// TIA Portal V17 export
// export: Created 2025-03-07T09:18:59.1372359Z, ExportSetting WithDefaults, DisplayName Totally Integrated Automation Portal, DisplayVersion V17 Update 8, DisplayName TIA Portal Openness, DisplayVersion V17 Update 8, DisplayName TIA Portal Version Control Interface, DisplayVersion V17, DisplayName SINAMICS Startdrive Advanced, DisplayVersion V17 SP2, DisplayName SINAMICS Startdrive G110M, G120, G120C, G120D, G120P, G115D, DisplayVersion V17 SP2, DisplayName SINAMICS Startdrive G130, G150, S120, S150, SINAMICS MV, S210, DisplayVersion V17 SP2, DisplayName STEP 7 Professional, DisplayVersion V17 Update 8, DisplayName SINUMERIK ONE STEP 7 Toolbox, DisplayVersion V17 Update 12, DisplayName SINUMERIK 840D sl STEP 7 Toolbox, DisplayVersion V17 Update 12, DisplayName STEP 7 Safety, DisplayVersion V17 Update 6, DisplayName WinCC Advanced, DisplayVersion V17 Update 8
FUNCTION "FC16017_METHOD_CALLS_U03_MEAS_STA_MEAS_B" : Void   // FC16017, LAD
{ S7_Optimized_Access := 'TRUE' }
VERSION : 0.1
// stored: AutoNumber false, IsIECCheckEnabled false, SetENOAutomatically false, UDAEnableTagReadback false
   VAR_TEMP
      AUX_WSTRING_PART_ID_MEAS_STA : WString;
      AUX_WCHARS : Array[0..63] of WChar;
      index : Int;
      AUX_ALARMS : Bool;
   END_VAR
   VAR_TEMP   // added for the SCL form of the ladder/FBD networks
      _w1 : Bool;
      _w2 : Bool;
   END_VAR
BEGIN

REGION Network 1 (SCL): TRANSFORM TO WCHARS
   FOR #index := 0 TO 63 DO
       #AUX_WCHARS[#index] := CHAR_TO_WCHAR("DB8000_PART_STATUS".UNIT_03.FIXTURE_1.PART_A.PART_ID[#index]);
   END_FOR;
END_REGION

REGION Network 2: TRANSFORM TO WSTRING
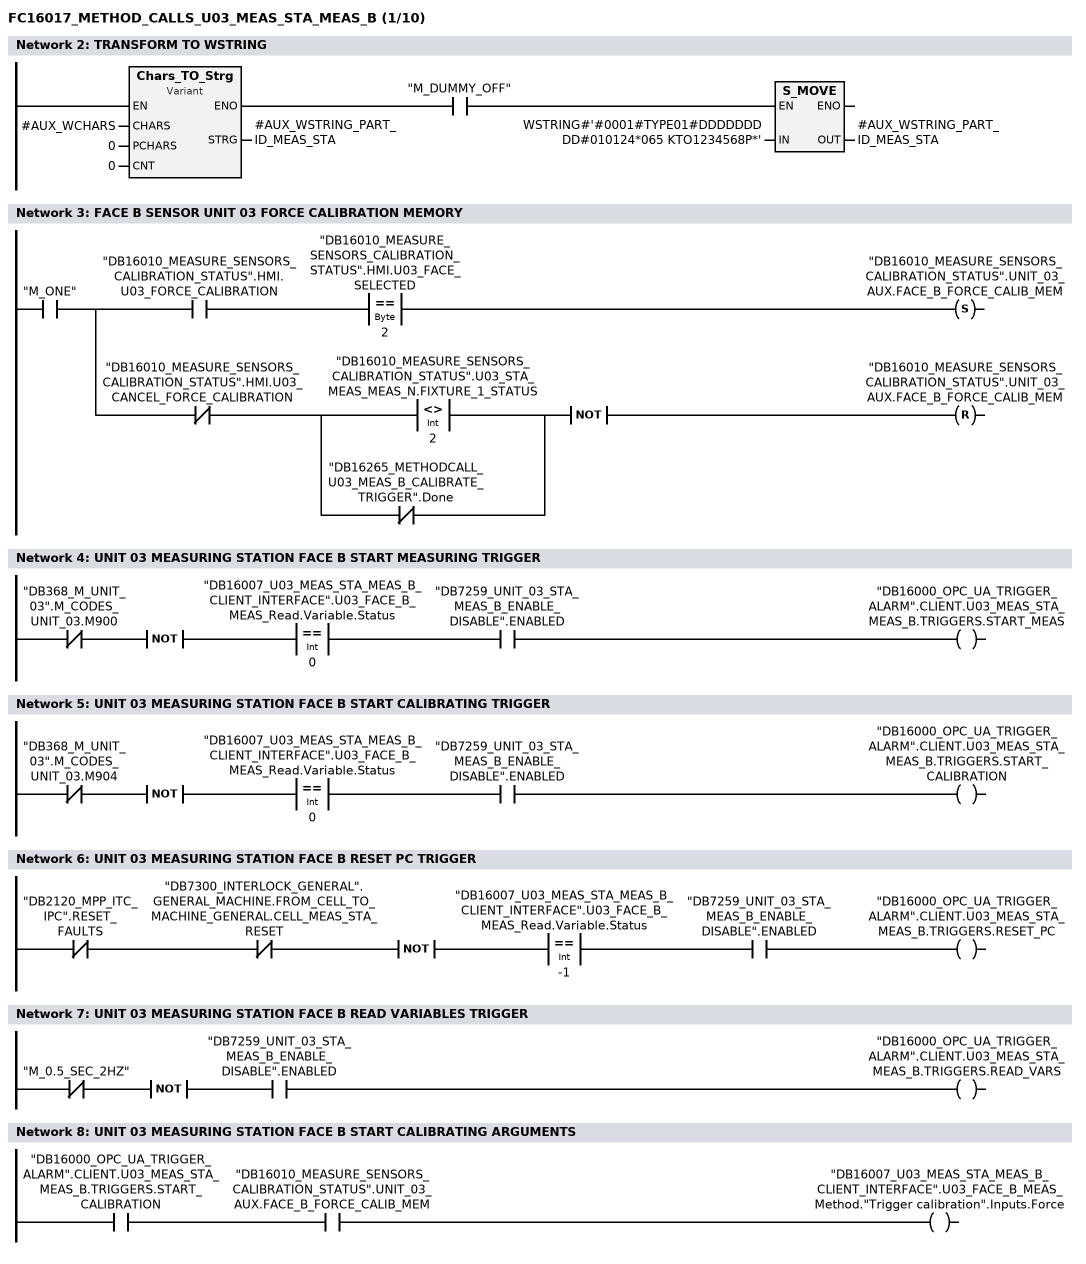
   RUNG wire#powerrail
      { S7_Templates := "[ptr_type := Variant, str_type := WString]" } Chars_TO_Strg(Chars := #AUX_WCHARS, pChars := 0, Cnt := 0, Strg => #AUX_WSTRING_PART_ID_MEAS_STA)
      Contact( "M_DUMMY_OFF" )
      S_Move(in := WSTRING#'#0001#TYPE01#DDDDDDDDD#010124*065 KTO1234568P*', out => #AUX_WSTRING_PART_ID_MEAS_STA)
   END_RUNG
   // the same network as SCL:
   Chars_TO_Strg(Chars := #AUX_WCHARS,
                 pChars := 0,
                 Cnt := 0,
                 Strg => #AUX_WSTRING_PART_ID_MEAS_STA,
                 ENO => #_w1);
   IF #_w1 AND "M_DUMMY_OFF" THEN
       #AUX_WSTRING_PART_ID_MEAS_STA := WSTRING#'#0001#TYPE01#DDDDDDDDD#010124*065 KTO1234568P*';
   END_IF;
END_REGION

REGION Network 3: FACE B SENSOR UNIT 03 FORCE CALIBRATION MEMORY
   RUNG wire#powerrail
      Contact( "M_ONE" )
      wire#w1
      Contact( "DB16010_MEASURE_SENSORS_CALIBRATION_STATUS".HMI.U03_FORCE_CALIBRATION )
      { S7_Templates := "SrcType := Byte" } EQ_Contact(in1 := "DB16010_MEASURE_SENSORS_CALIBRATION_STATUS".HMI.U03_FACE_SELECTED, in2 := 2)
      S_Coil( "DB16010_MEASURE_SENSORS_CALIBRATION_STATUS".UNIT_03_AUX.FACE_B_FORCE_CALIB_MEM )
   END_RUNG
   RUNG wire#w1
      I_Contact( "DB16010_MEASURE_SENSORS_CALIBRATION_STATUS".HMI.U03_CANCEL_FORCE_CALIBRATION )
      wire#w2
      { S7_Templates := "SrcType := Int" } NE_Contact(in1 := "DB16010_MEASURE_SENSORS_CALIBRATION_STATUS".U03_STA_MEAS_MEAS_N.FIXTURE_1_STATUS, in2 := 2)
      wire#w3
      Not()
      R_Coil( "DB16010_MEASURE_SENSORS_CALIBRATION_STATUS".UNIT_03_AUX.FACE_B_FORCE_CALIB_MEM )
   END_RUNG
   RUNG wire#w2
      I_Contact( "DB16265_METHODCALL_U03_MEAS_B_CALIBRATE_TRIGGER".Done )
   END_RUNG wire#w3
   // the same network as SCL:
   IF "M_ONE" AND "DB16010_MEASURE_SENSORS_CALIBRATION_STATUS".HMI.U03_FORCE_CALIBRATION AND ("DB16010_MEASURE_SENSORS_CALIBRATION_STATUS".HMI.U03_FACE_SELECTED = 2) THEN
       "DB16010_MEASURE_SENSORS_CALIBRATION_STATUS".UNIT_03_AUX.FACE_B_FORCE_CALIB_MEM := TRUE;
   END_IF;
   IF NOT ("M_ONE" AND NOT "DB16010_MEASURE_SENSORS_CALIBRATION_STATUS".HMI.U03_CANCEL_FORCE_CALIBRATION AND (("DB16010_MEASURE_SENSORS_CALIBRATION_STATUS".U03_STA_MEAS_MEAS_N.FIXTURE_1_STATUS <> 2) OR NOT "DB16265_METHODCALL_U03_MEAS_B_CALIBRATE_TRIGGER".Done)) THEN
       "DB16010_MEASURE_SENSORS_CALIBRATION_STATUS".UNIT_03_AUX.FACE_B_FORCE_CALIB_MEM := FALSE;
   END_IF;
END_REGION

REGION Network 4: UNIT 03 MEASURING STATION FACE B START MEASURING TRIGGER
   RUNG wire#powerrail
      I_Contact( "DB368_M_UNIT_03".M_CODES_UNIT_03.M900 )
      Not()
      { S7_Templates := "SrcType := Int" } EQ_Contact(in1 := "DB16007_U03_MEAS_STA_MEAS_B_CLIENT_INTERFACE".U03_FACE_B_MEAS_Read.Variable.Status, in2 := 0)
      Contact( "DB7259_UNIT_03_STA_MEAS_B_ENABLE_DISABLE".ENABLED )
      Coil( "DB16000_OPC_UA_TRIGGER_ALARM".CLIENT.U03_MEAS_STA_MEAS_B.TRIGGERS.START_MEAS )
   END_RUNG
   // the same network as SCL:
   "DB16000_OPC_UA_TRIGGER_ALARM".CLIENT.U03_MEAS_STA_MEAS_B.TRIGGERS.START_MEAS := NOT (NOT "DB368_M_UNIT_03".M_CODES_UNIT_03.M900) AND ("DB16007_U03_MEAS_STA_MEAS_B_CLIENT_INTERFACE".U03_FACE_B_MEAS_Read.Variable.Status = 0) AND "DB7259_UNIT_03_STA_MEAS_B_ENABLE_DISABLE".ENABLED;
END_REGION

REGION Network 5: UNIT 03 MEASURING STATION FACE B START CALIBRATING TRIGGER
   RUNG wire#powerrail
      I_Contact( "DB368_M_UNIT_03".M_CODES_UNIT_03.M904 )
      Not()
      { S7_Templates := "SrcType := Int" } EQ_Contact(in1 := "DB16007_U03_MEAS_STA_MEAS_B_CLIENT_INTERFACE".U03_FACE_B_MEAS_Read.Variable.Status, in2 := 0)
      Contact( "DB7259_UNIT_03_STA_MEAS_B_ENABLE_DISABLE".ENABLED )
      Coil( "DB16000_OPC_UA_TRIGGER_ALARM".CLIENT.U03_MEAS_STA_MEAS_B.TRIGGERS.START_CALIBRATION )
   END_RUNG
   // the same network as SCL:
   "DB16000_OPC_UA_TRIGGER_ALARM".CLIENT.U03_MEAS_STA_MEAS_B.TRIGGERS.START_CALIBRATION := NOT (NOT "DB368_M_UNIT_03".M_CODES_UNIT_03.M904) AND ("DB16007_U03_MEAS_STA_MEAS_B_CLIENT_INTERFACE".U03_FACE_B_MEAS_Read.Variable.Status = 0) AND "DB7259_UNIT_03_STA_MEAS_B_ENABLE_DISABLE".ENABLED;
END_REGION

REGION Network 6: UNIT 03 MEASURING STATION FACE B RESET PC TRIGGER
   RUNG wire#powerrail
      I_Contact( "DB2120_MPP_ITC_IPC".RESET_FAULTS )
      I_Contact( "DB7300_INTERLOCK_GENERAL".GENERAL_MACHINE.FROM_CELL_TO_MACHINE_GENERAL.CELL_MEAS_STA_RESET )
      Not()
      { S7_Templates := "SrcType := Int" } EQ_Contact(in1 := "DB16007_U03_MEAS_STA_MEAS_B_CLIENT_INTERFACE".U03_FACE_B_MEAS_Read.Variable.Status, in2 := -1)
      Contact( "DB7259_UNIT_03_STA_MEAS_B_ENABLE_DISABLE".ENABLED )
      Coil( "DB16000_OPC_UA_TRIGGER_ALARM".CLIENT.U03_MEAS_STA_MEAS_B.TRIGGERS.RESET_PC )
   END_RUNG
   // the same network as SCL:
   "DB16000_OPC_UA_TRIGGER_ALARM".CLIENT.U03_MEAS_STA_MEAS_B.TRIGGERS.RESET_PC := NOT (NOT "DB2120_MPP_ITC_IPC".RESET_FAULTS AND NOT "DB7300_INTERLOCK_GENERAL".GENERAL_MACHINE.FROM_CELL_TO_MACHINE_GENERAL.CELL_MEAS_STA_RESET) AND ("DB16007_U03_MEAS_STA_MEAS_B_CLIENT_INTERFACE".U03_FACE_B_MEAS_Read.Variable.Status = (-1)) AND "DB7259_UNIT_03_STA_MEAS_B_ENABLE_DISABLE".ENABLED;
END_REGION

REGION Network 7: UNIT 03 MEASURING STATION FACE B READ VARIABLES TRIGGER
   RUNG wire#powerrail
      I_Contact( "M_0.5_SEC_2HZ" )
      Not()
      Contact( "DB7259_UNIT_03_STA_MEAS_B_ENABLE_DISABLE".ENABLED )
      Coil( "DB16000_OPC_UA_TRIGGER_ALARM".CLIENT.U03_MEAS_STA_MEAS_B.TRIGGERS.READ_VARS )
   END_RUNG
   // the same network as SCL:
   "DB16000_OPC_UA_TRIGGER_ALARM".CLIENT.U03_MEAS_STA_MEAS_B.TRIGGERS.READ_VARS := NOT (NOT "M_0.5_SEC_2HZ") AND "DB7259_UNIT_03_STA_MEAS_B_ENABLE_DISABLE".ENABLED;
END_REGION

REGION Network 8: UNIT 03 MEASURING STATION FACE B START CALIBRATING ARGUMENTS
   RUNG wire#powerrail
      Contact( "DB16000_OPC_UA_TRIGGER_ALARM".CLIENT.U03_MEAS_STA_MEAS_B.TRIGGERS.START_CALIBRATION )
      Contact( "DB16010_MEASURE_SENSORS_CALIBRATION_STATUS".UNIT_03_AUX.FACE_B_FORCE_CALIB_MEM )
      Coil( "DB16007_U03_MEAS_STA_MEAS_B_CLIENT_INTERFACE".U03_FACE_B_MEAS_Method."Trigger calibration".Inputs.Force )
   END_RUNG
   // the same network as SCL:
   "DB16007_U03_MEAS_STA_MEAS_B_CLIENT_INTERFACE".U03_FACE_B_MEAS_Method."Trigger calibration".Inputs.Force := "DB16000_OPC_UA_TRIGGER_ALARM".CLIENT.U03_MEAS_STA_MEAS_B.TRIGGERS.START_CALIBRATION AND "DB16010_MEASURE_SENSORS_CALIBRATION_STATUS".UNIT_03_AUX.FACE_B_FORCE_CALIB_MEM;
END_REGION

REGION Network 9: UNIT 03 MEASURING STATION FACE B START MEASURING TRIGGER CALL
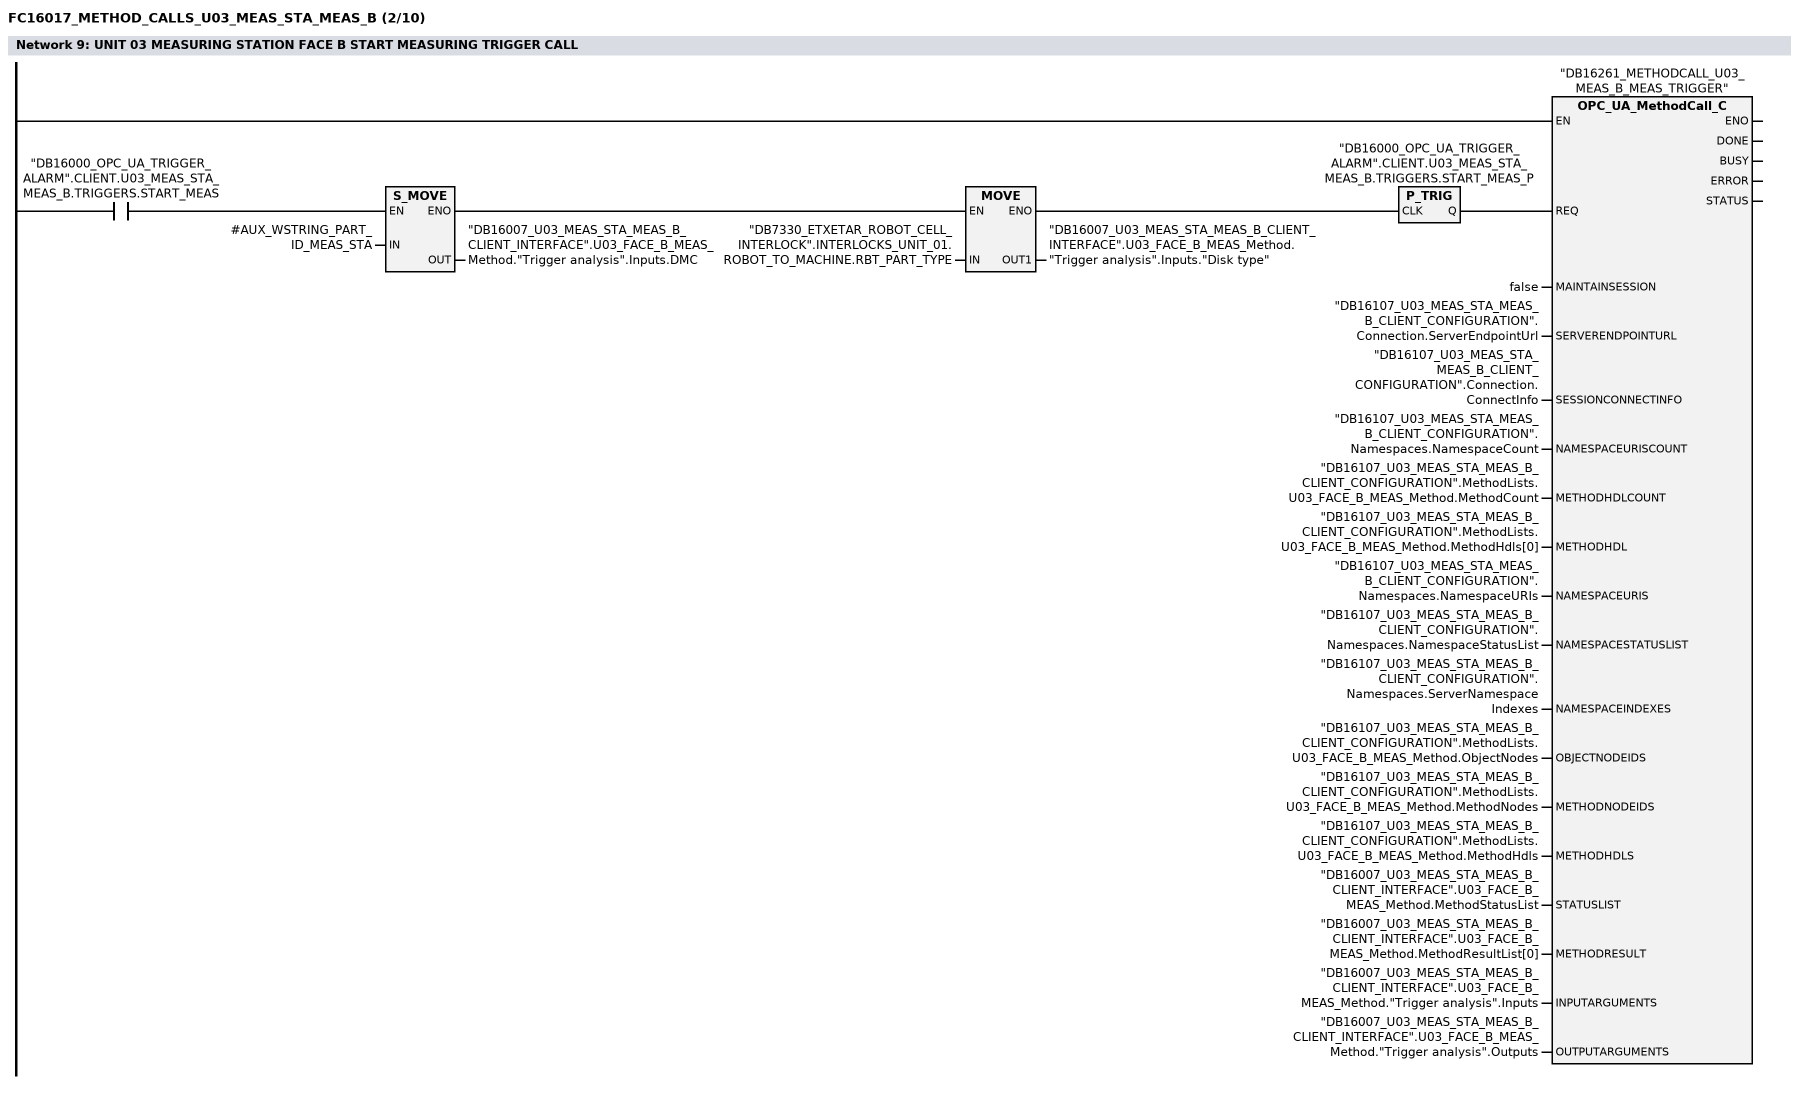
   RUNG wire#powerrail
      "DB16261_METHODCALL_U03_MEAS_B_MEAS_TRIGGER".OPC_UA_MethodCall_C(REQ := wire#w1, MaintainSession := false, ServerEndpointUrl := "DB16107_U03_MEAS_STA_MEAS_B_CLIENT_CONFIGURATION".Connection.ServerEndpointUrl, SessionConnectInfo := "DB16107_U03_MEAS_STA_MEAS_B_CLIENT_CONFIGURATION".Connection.ConnectInfo, NamespaceUrisCount := "DB16107_U03_MEAS_STA_MEAS_B_CLIENT_CONFIGURATION".Namespaces.NamespaceCount, MethodHdlCount := "DB16107_U03_MEAS_STA_MEAS_B_CLIENT_CONFIGURATION".MethodLists.U03_FACE_B_MEAS_Method.MethodCount, MethodHdl := "DB16107_U03_MEAS_STA_MEAS_B_CLIENT_CONFIGURATION".MethodLists.U03_FACE_B_MEAS_Method.MethodHdls[0], NamespaceUris := "DB16107_U03_MEAS_STA_MEAS_B_CLIENT_CONFIGURATION".Namespaces.NamespaceURIs, NamespaceStatusList := "DB16107_U03_MEAS_STA_MEAS_B_CLIENT_CONFIGURATION".Namespaces.NamespaceStatusList, NamespaceIndexes := "DB16107_U03_MEAS_STA_MEAS_B_CLIENT_CONFIGURATION".Namespaces.ServerNamespaceIndexes, ObjectNodeIDs := "DB16107_U03_MEAS_STA_MEAS_B_CLIENT_CONFIGURATION".MethodLists.U03_FACE_B_MEAS_Method.ObjectNodes, MethodNodeIDs := "DB16107_U03_MEAS_STA_MEAS_B_CLIENT_CONFIGURATION".MethodLists.U03_FACE_B_MEAS_Method.MethodNodes, MethodHdls := "DB16107_U03_MEAS_STA_MEAS_B_CLIENT_CONFIGURATION".MethodLists.U03_FACE_B_MEAS_Method.MethodHdls, StatusList := "DB16007_U03_MEAS_STA_MEAS_B_CLIENT_INTERFACE".U03_FACE_B_MEAS_Method.MethodStatusList, MethodResult := "DB16007_U03_MEAS_STA_MEAS_B_CLIENT_INTERFACE".U03_FACE_B_MEAS_Method.MethodResultList[0], InputArguments := "DB16007_U03_MEAS_STA_MEAS_B_CLIENT_INTERFACE".U03_FACE_B_MEAS_Method."Trigger analysis".Inputs, OutputArguments := "DB16007_U03_MEAS_STA_MEAS_B_CLIENT_INTERFACE".U03_FACE_B_MEAS_Method."Trigger analysis".Outputs, Done =>, Busy =>, Error =>, Status =>)
   END_RUNG
   RUNG wire#powerrail
      Contact( "DB16000_OPC_UA_TRIGGER_ALARM".CLIENT.U03_MEAS_STA_MEAS_B.TRIGGERS.START_MEAS )
      S_Move(in := #AUX_WSTRING_PART_ID_MEAS_STA, out => "DB16007_U03_MEAS_STA_MEAS_B_CLIENT_INTERFACE".U03_FACE_B_MEAS_Method."Trigger analysis".Inputs.DMC)
      Move(in := "DB7330_ETXETAR_ROBOT_CELL_INTERLOCK".INTERLOCKS_UNIT_01.ROBOT_TO_MACHINE.RBT_PART_TYPE, out1 => "DB16007_U03_MEAS_STA_MEAS_B_CLIENT_INTERFACE".U03_FACE_B_MEAS_Method."Trigger analysis".Inputs."Disk type")
      P_Trig( "DB16000_OPC_UA_TRIGGER_ALARM".CLIENT.U03_MEAS_STA_MEAS_B.TRIGGERS.START_MEAS_P )
   END_RUNG wire#w1
   // the same network as SCL:
   IF "DB16000_OPC_UA_TRIGGER_ALARM".CLIENT.U03_MEAS_STA_MEAS_B.TRIGGERS.START_MEAS THEN
       "DB16007_U03_MEAS_STA_MEAS_B_CLIENT_INTERFACE".U03_FACE_B_MEAS_Method."Trigger analysis".Inputs.DMC := #AUX_WSTRING_PART_ID_MEAS_STA;
       "DB16007_U03_MEAS_STA_MEAS_B_CLIENT_INTERFACE".U03_FACE_B_MEAS_Method."Trigger analysis".Inputs."Disk type" := "DB7330_ETXETAR_ROBOT_CELL_INTERLOCK".INTERLOCKS_UNIT_01.ROBOT_TO_MACHINE.RBT_PART_TYPE;
   END_IF;
   #_w1 := "DB16000_OPC_UA_TRIGGER_ALARM".CLIENT.U03_MEAS_STA_MEAS_B.TRIGGERS.START_MEAS AND NOT "DB16000_OPC_UA_TRIGGER_ALARM".CLIENT.U03_MEAS_STA_MEAS_B.TRIGGERS.START_MEAS_P;   // rising edge
   "DB16000_OPC_UA_TRIGGER_ALARM".CLIENT.U03_MEAS_STA_MEAS_B.TRIGGERS.START_MEAS_P := "DB16000_OPC_UA_TRIGGER_ALARM".CLIENT.U03_MEAS_STA_MEAS_B.TRIGGERS.START_MEAS;
   "DB16261_METHODCALL_U03_MEAS_B_MEAS_TRIGGER"(REQ := #_w1,   // OPC_UA_MethodCall_C
                           MaintainSession := false,
                           ServerEndpointUrl := "DB16107_U03_MEAS_STA_MEAS_B_CLIENT_CONFIGURATION".Connection.ServerEndpointUrl,
                           SessionConnectInfo := "DB16107_U03_MEAS_STA_MEAS_B_CLIENT_CONFIGURATION".Connection.ConnectInfo,
                           NamespaceUrisCount := "DB16107_U03_MEAS_STA_MEAS_B_CLIENT_CONFIGURATION".Namespaces.NamespaceCount,
                           MethodHdlCount := "DB16107_U03_MEAS_STA_MEAS_B_CLIENT_CONFIGURATION".MethodLists.U03_FACE_B_MEAS_Method.MethodCount,
                           MethodHdl := "DB16107_U03_MEAS_STA_MEAS_B_CLIENT_CONFIGURATION".MethodLists.U03_FACE_B_MEAS_Method.MethodHdls[0],
                           NamespaceUris := "DB16107_U03_MEAS_STA_MEAS_B_CLIENT_CONFIGURATION".Namespaces.NamespaceURIs,
                           NamespaceStatusList := "DB16107_U03_MEAS_STA_MEAS_B_CLIENT_CONFIGURATION".Namespaces.NamespaceStatusList,
                           NamespaceIndexes := "DB16107_U03_MEAS_STA_MEAS_B_CLIENT_CONFIGURATION".Namespaces.ServerNamespaceIndexes,
                           ObjectNodeIDs := "DB16107_U03_MEAS_STA_MEAS_B_CLIENT_CONFIGURATION".MethodLists.U03_FACE_B_MEAS_Method.ObjectNodes,
                           MethodNodeIDs := "DB16107_U03_MEAS_STA_MEAS_B_CLIENT_CONFIGURATION".MethodLists.U03_FACE_B_MEAS_Method.MethodNodes,
                           MethodHdls := "DB16107_U03_MEAS_STA_MEAS_B_CLIENT_CONFIGURATION".MethodLists.U03_FACE_B_MEAS_Method.MethodHdls,
                           StatusList := "DB16007_U03_MEAS_STA_MEAS_B_CLIENT_INTERFACE".U03_FACE_B_MEAS_Method.MethodStatusList,
                           MethodResult := "DB16007_U03_MEAS_STA_MEAS_B_CLIENT_INTERFACE".U03_FACE_B_MEAS_Method.MethodResultList[0],
                           InputArguments := "DB16007_U03_MEAS_STA_MEAS_B_CLIENT_INTERFACE".U03_FACE_B_MEAS_Method."Trigger analysis".Inputs,
                           OutputArguments := "DB16007_U03_MEAS_STA_MEAS_B_CLIENT_INTERFACE".U03_FACE_B_MEAS_Method."Trigger analysis".Outputs);
END_REGION

REGION Network 10: UNIT 03 MEASURING STATION FACE B START CALIBRATING TRIGGER CALL
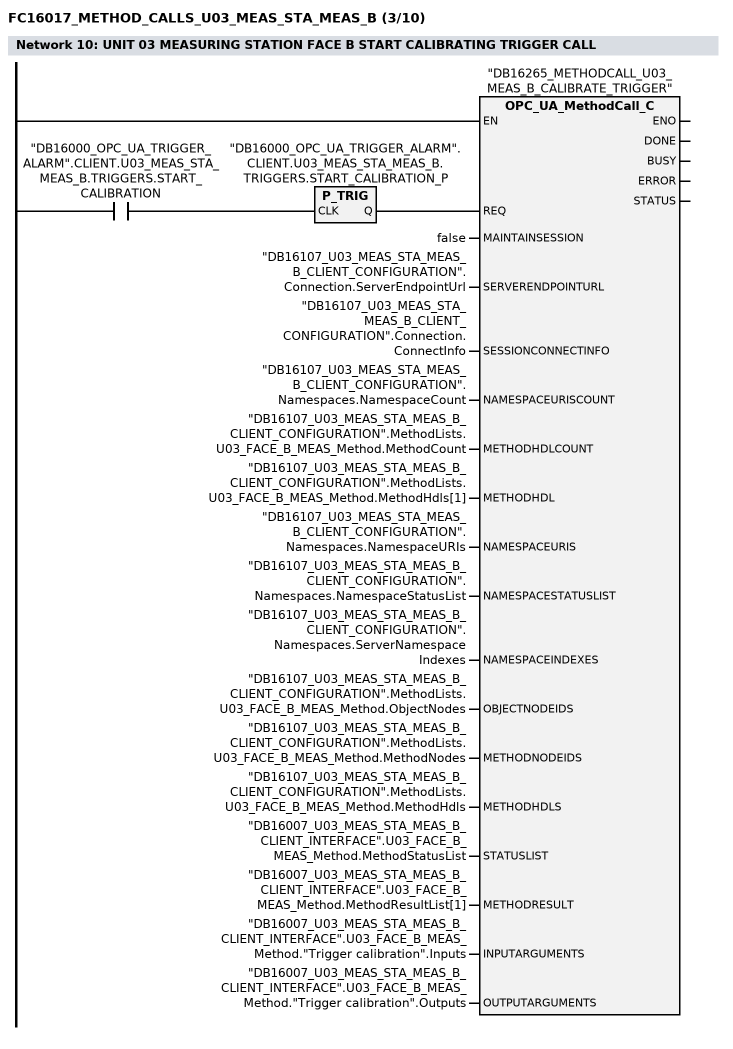
   RUNG wire#powerrail
      "DB16265_METHODCALL_U03_MEAS_B_CALIBRATE_TRIGGER".OPC_UA_MethodCall_C(REQ := wire#w1, MaintainSession := false, ServerEndpointUrl := "DB16107_U03_MEAS_STA_MEAS_B_CLIENT_CONFIGURATION".Connection.ServerEndpointUrl, SessionConnectInfo := "DB16107_U03_MEAS_STA_MEAS_B_CLIENT_CONFIGURATION".Connection.ConnectInfo, NamespaceUrisCount := "DB16107_U03_MEAS_STA_MEAS_B_CLIENT_CONFIGURATION".Namespaces.NamespaceCount, MethodHdlCount := "DB16107_U03_MEAS_STA_MEAS_B_CLIENT_CONFIGURATION".MethodLists.U03_FACE_B_MEAS_Method.MethodCount, MethodHdl := "DB16107_U03_MEAS_STA_MEAS_B_CLIENT_CONFIGURATION".MethodLists.U03_FACE_B_MEAS_Method.MethodHdls[1], NamespaceUris := "DB16107_U03_MEAS_STA_MEAS_B_CLIENT_CONFIGURATION".Namespaces.NamespaceURIs, NamespaceStatusList := "DB16107_U03_MEAS_STA_MEAS_B_CLIENT_CONFIGURATION".Namespaces.NamespaceStatusList, NamespaceIndexes := "DB16107_U03_MEAS_STA_MEAS_B_CLIENT_CONFIGURATION".Namespaces.ServerNamespaceIndexes, ObjectNodeIDs := "DB16107_U03_MEAS_STA_MEAS_B_CLIENT_CONFIGURATION".MethodLists.U03_FACE_B_MEAS_Method.ObjectNodes, MethodNodeIDs := "DB16107_U03_MEAS_STA_MEAS_B_CLIENT_CONFIGURATION".MethodLists.U03_FACE_B_MEAS_Method.MethodNodes, MethodHdls := "DB16107_U03_MEAS_STA_MEAS_B_CLIENT_CONFIGURATION".MethodLists.U03_FACE_B_MEAS_Method.MethodHdls, StatusList := "DB16007_U03_MEAS_STA_MEAS_B_CLIENT_INTERFACE".U03_FACE_B_MEAS_Method.MethodStatusList, MethodResult := "DB16007_U03_MEAS_STA_MEAS_B_CLIENT_INTERFACE".U03_FACE_B_MEAS_Method.MethodResultList[1], InputArguments := "DB16007_U03_MEAS_STA_MEAS_B_CLIENT_INTERFACE".U03_FACE_B_MEAS_Method."Trigger calibration".Inputs, OutputArguments := "DB16007_U03_MEAS_STA_MEAS_B_CLIENT_INTERFACE".U03_FACE_B_MEAS_Method."Trigger calibration".Outputs, Done =>, Busy =>, Error =>, Status =>)
   END_RUNG
   RUNG wire#powerrail
      Contact( "DB16000_OPC_UA_TRIGGER_ALARM".CLIENT.U03_MEAS_STA_MEAS_B.TRIGGERS.START_CALIBRATION )
      P_Trig( "DB16000_OPC_UA_TRIGGER_ALARM".CLIENT.U03_MEAS_STA_MEAS_B.TRIGGERS.START_CALIBRATION_P )
   END_RUNG wire#w1
   // the same network as SCL:
   #_w1 := "DB16000_OPC_UA_TRIGGER_ALARM".CLIENT.U03_MEAS_STA_MEAS_B.TRIGGERS.START_CALIBRATION AND NOT "DB16000_OPC_UA_TRIGGER_ALARM".CLIENT.U03_MEAS_STA_MEAS_B.TRIGGERS.START_CALIBRATION_P;   // rising edge
   "DB16000_OPC_UA_TRIGGER_ALARM".CLIENT.U03_MEAS_STA_MEAS_B.TRIGGERS.START_CALIBRATION_P := "DB16000_OPC_UA_TRIGGER_ALARM".CLIENT.U03_MEAS_STA_MEAS_B.TRIGGERS.START_CALIBRATION;
   "DB16265_METHODCALL_U03_MEAS_B_CALIBRATE_TRIGGER"(REQ := #_w1,   // OPC_UA_MethodCall_C
                           MaintainSession := false,
                           ServerEndpointUrl := "DB16107_U03_MEAS_STA_MEAS_B_CLIENT_CONFIGURATION".Connection.ServerEndpointUrl,
                           SessionConnectInfo := "DB16107_U03_MEAS_STA_MEAS_B_CLIENT_CONFIGURATION".Connection.ConnectInfo,
                           NamespaceUrisCount := "DB16107_U03_MEAS_STA_MEAS_B_CLIENT_CONFIGURATION".Namespaces.NamespaceCount,
                           MethodHdlCount := "DB16107_U03_MEAS_STA_MEAS_B_CLIENT_CONFIGURATION".MethodLists.U03_FACE_B_MEAS_Method.MethodCount,
                           MethodHdl := "DB16107_U03_MEAS_STA_MEAS_B_CLIENT_CONFIGURATION".MethodLists.U03_FACE_B_MEAS_Method.MethodHdls[1],
                           NamespaceUris := "DB16107_U03_MEAS_STA_MEAS_B_CLIENT_CONFIGURATION".Namespaces.NamespaceURIs,
                           NamespaceStatusList := "DB16107_U03_MEAS_STA_MEAS_B_CLIENT_CONFIGURATION".Namespaces.NamespaceStatusList,
                           NamespaceIndexes := "DB16107_U03_MEAS_STA_MEAS_B_CLIENT_CONFIGURATION".Namespaces.ServerNamespaceIndexes,
                           ObjectNodeIDs := "DB16107_U03_MEAS_STA_MEAS_B_CLIENT_CONFIGURATION".MethodLists.U03_FACE_B_MEAS_Method.ObjectNodes,
                           MethodNodeIDs := "DB16107_U03_MEAS_STA_MEAS_B_CLIENT_CONFIGURATION".MethodLists.U03_FACE_B_MEAS_Method.MethodNodes,
                           MethodHdls := "DB16107_U03_MEAS_STA_MEAS_B_CLIENT_CONFIGURATION".MethodLists.U03_FACE_B_MEAS_Method.MethodHdls,
                           StatusList := "DB16007_U03_MEAS_STA_MEAS_B_CLIENT_INTERFACE".U03_FACE_B_MEAS_Method.MethodStatusList,
                           MethodResult := "DB16007_U03_MEAS_STA_MEAS_B_CLIENT_INTERFACE".U03_FACE_B_MEAS_Method.MethodResultList[1],
                           InputArguments := "DB16007_U03_MEAS_STA_MEAS_B_CLIENT_INTERFACE".U03_FACE_B_MEAS_Method."Trigger calibration".Inputs,
                           OutputArguments := "DB16007_U03_MEAS_STA_MEAS_B_CLIENT_INTERFACE".U03_FACE_B_MEAS_Method."Trigger calibration".Outputs);
END_REGION

REGION Network 11: UNIT 03 MEASURING STATION FACE B RESET PC TRIGGER CALL
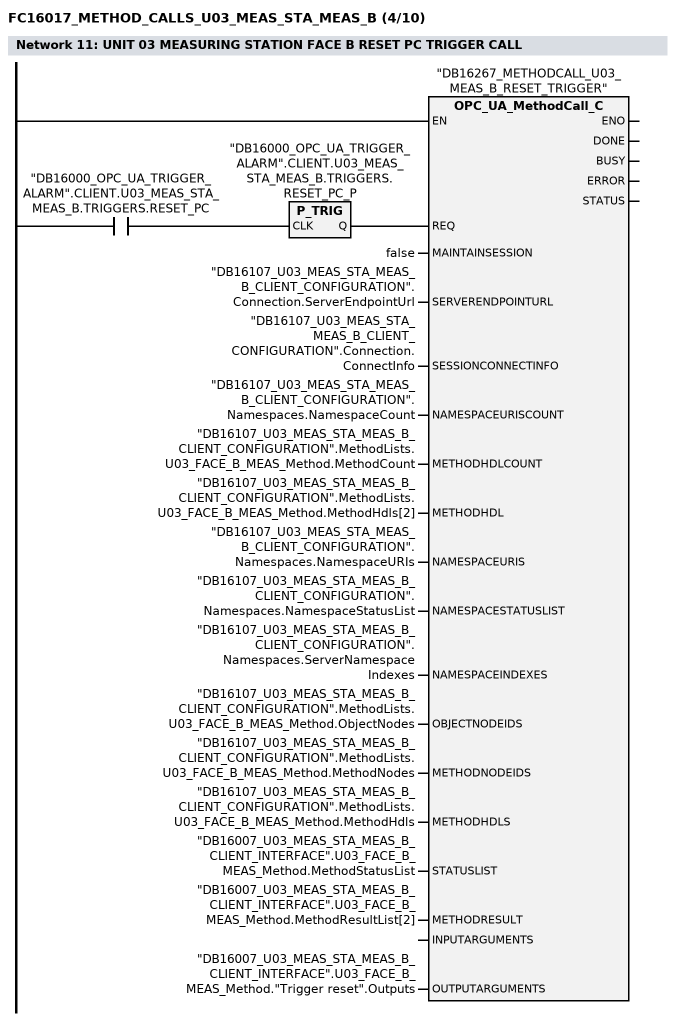
   RUNG wire#powerrail
      "DB16267_METHODCALL_U03_MEAS_B_RESET_TRIGGER".OPC_UA_MethodCall_C(REQ := wire#w1, MaintainSession := false, ServerEndpointUrl := "DB16107_U03_MEAS_STA_MEAS_B_CLIENT_CONFIGURATION".Connection.ServerEndpointUrl, SessionConnectInfo := "DB16107_U03_MEAS_STA_MEAS_B_CLIENT_CONFIGURATION".Connection.ConnectInfo, NamespaceUrisCount := "DB16107_U03_MEAS_STA_MEAS_B_CLIENT_CONFIGURATION".Namespaces.NamespaceCount, MethodHdlCount := "DB16107_U03_MEAS_STA_MEAS_B_CLIENT_CONFIGURATION".MethodLists.U03_FACE_B_MEAS_Method.MethodCount, MethodHdl := "DB16107_U03_MEAS_STA_MEAS_B_CLIENT_CONFIGURATION".MethodLists.U03_FACE_B_MEAS_Method.MethodHdls[2], NamespaceUris := "DB16107_U03_MEAS_STA_MEAS_B_CLIENT_CONFIGURATION".Namespaces.NamespaceURIs, NamespaceStatusList := "DB16107_U03_MEAS_STA_MEAS_B_CLIENT_CONFIGURATION".Namespaces.NamespaceStatusList, NamespaceIndexes := "DB16107_U03_MEAS_STA_MEAS_B_CLIENT_CONFIGURATION".Namespaces.ServerNamespaceIndexes, ObjectNodeIDs := "DB16107_U03_MEAS_STA_MEAS_B_CLIENT_CONFIGURATION".MethodLists.U03_FACE_B_MEAS_Method.ObjectNodes, MethodNodeIDs := "DB16107_U03_MEAS_STA_MEAS_B_CLIENT_CONFIGURATION".MethodLists.U03_FACE_B_MEAS_Method.MethodNodes, MethodHdls := "DB16107_U03_MEAS_STA_MEAS_B_CLIENT_CONFIGURATION".MethodLists.U03_FACE_B_MEAS_Method.MethodHdls, StatusList := "DB16007_U03_MEAS_STA_MEAS_B_CLIENT_INTERFACE".U03_FACE_B_MEAS_Method.MethodStatusList, MethodResult := "DB16007_U03_MEAS_STA_MEAS_B_CLIENT_INTERFACE".U03_FACE_B_MEAS_Method.MethodResultList[2], InputArguments :=, OutputArguments := "DB16007_U03_MEAS_STA_MEAS_B_CLIENT_INTERFACE".U03_FACE_B_MEAS_Method."Trigger reset".Outputs, Done =>, Busy =>, Error =>, Status =>)
   END_RUNG
   RUNG wire#powerrail
      Contact( "DB16000_OPC_UA_TRIGGER_ALARM".CLIENT.U03_MEAS_STA_MEAS_B.TRIGGERS.RESET_PC )
      P_Trig( "DB16000_OPC_UA_TRIGGER_ALARM".CLIENT.U03_MEAS_STA_MEAS_B.TRIGGERS.RESET_PC_P )
   END_RUNG wire#w1
   // the same network as SCL:
   #_w1 := "DB16000_OPC_UA_TRIGGER_ALARM".CLIENT.U03_MEAS_STA_MEAS_B.TRIGGERS.RESET_PC AND NOT "DB16000_OPC_UA_TRIGGER_ALARM".CLIENT.U03_MEAS_STA_MEAS_B.TRIGGERS.RESET_PC_P;   // rising edge
   "DB16000_OPC_UA_TRIGGER_ALARM".CLIENT.U03_MEAS_STA_MEAS_B.TRIGGERS.RESET_PC_P := "DB16000_OPC_UA_TRIGGER_ALARM".CLIENT.U03_MEAS_STA_MEAS_B.TRIGGERS.RESET_PC;
   "DB16267_METHODCALL_U03_MEAS_B_RESET_TRIGGER"(REQ := #_w1,   // OPC_UA_MethodCall_C
                           MaintainSession := false,
                           ServerEndpointUrl := "DB16107_U03_MEAS_STA_MEAS_B_CLIENT_CONFIGURATION".Connection.ServerEndpointUrl,
                           SessionConnectInfo := "DB16107_U03_MEAS_STA_MEAS_B_CLIENT_CONFIGURATION".Connection.ConnectInfo,
                           NamespaceUrisCount := "DB16107_U03_MEAS_STA_MEAS_B_CLIENT_CONFIGURATION".Namespaces.NamespaceCount,
                           MethodHdlCount := "DB16107_U03_MEAS_STA_MEAS_B_CLIENT_CONFIGURATION".MethodLists.U03_FACE_B_MEAS_Method.MethodCount,
                           MethodHdl := "DB16107_U03_MEAS_STA_MEAS_B_CLIENT_CONFIGURATION".MethodLists.U03_FACE_B_MEAS_Method.MethodHdls[2],
                           NamespaceUris := "DB16107_U03_MEAS_STA_MEAS_B_CLIENT_CONFIGURATION".Namespaces.NamespaceURIs,
                           NamespaceStatusList := "DB16107_U03_MEAS_STA_MEAS_B_CLIENT_CONFIGURATION".Namespaces.NamespaceStatusList,
                           NamespaceIndexes := "DB16107_U03_MEAS_STA_MEAS_B_CLIENT_CONFIGURATION".Namespaces.ServerNamespaceIndexes,
                           ObjectNodeIDs := "DB16107_U03_MEAS_STA_MEAS_B_CLIENT_CONFIGURATION".MethodLists.U03_FACE_B_MEAS_Method.ObjectNodes,
                           MethodNodeIDs := "DB16107_U03_MEAS_STA_MEAS_B_CLIENT_CONFIGURATION".MethodLists.U03_FACE_B_MEAS_Method.MethodNodes,
                           MethodHdls := "DB16107_U03_MEAS_STA_MEAS_B_CLIENT_CONFIGURATION".MethodLists.U03_FACE_B_MEAS_Method.MethodHdls,
                           StatusList := "DB16007_U03_MEAS_STA_MEAS_B_CLIENT_INTERFACE".U03_FACE_B_MEAS_Method.MethodStatusList,
                           MethodResult := "DB16007_U03_MEAS_STA_MEAS_B_CLIENT_INTERFACE".U03_FACE_B_MEAS_Method.MethodResultList[2],
                           OutputArguments := "DB16007_U03_MEAS_STA_MEAS_B_CLIENT_INTERFACE".U03_FACE_B_MEAS_Method."Trigger reset".Outputs);
END_REGION

REGION Network 12: UNIT 03 MEASURING STATION FACE B READ VARIABLES TRIGGER CALL
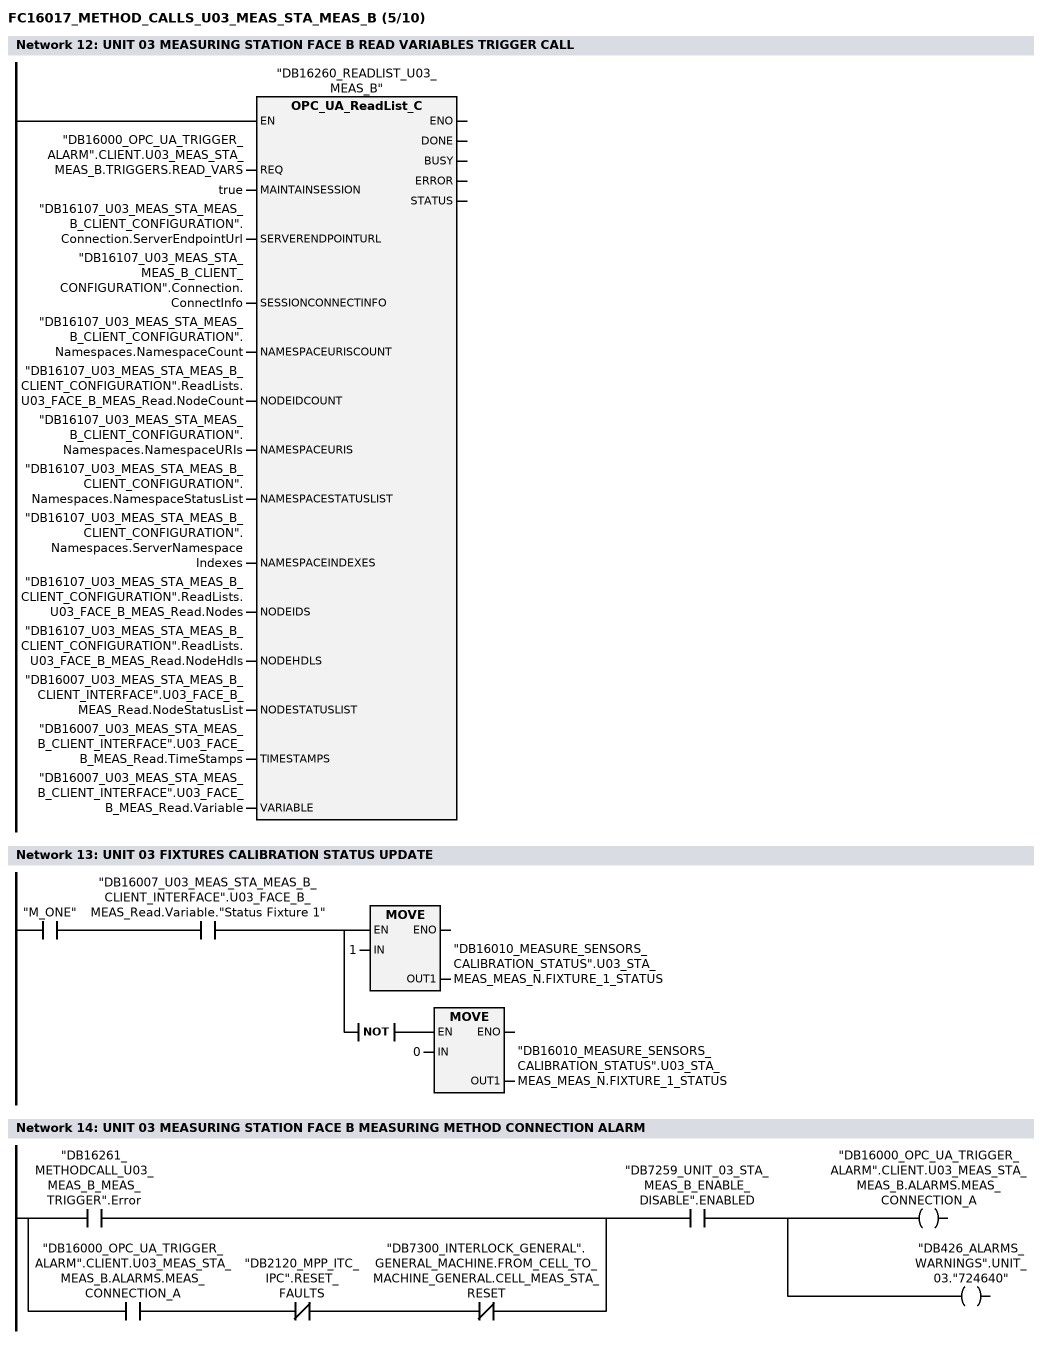
   RUNG wire#powerrail
      "DB16260_READLIST_U03_MEAS_B".OPC_UA_ReadList_C(REQ := "DB16000_OPC_UA_TRIGGER_ALARM".CLIENT.U03_MEAS_STA_MEAS_B.TRIGGERS.READ_VARS, MaintainSession := true, ServerEndpointUrl := "DB16107_U03_MEAS_STA_MEAS_B_CLIENT_CONFIGURATION".Connection.ServerEndpointUrl, SessionConnectInfo := "DB16107_U03_MEAS_STA_MEAS_B_CLIENT_CONFIGURATION".Connection.ConnectInfo, NamespaceUrisCount := "DB16107_U03_MEAS_STA_MEAS_B_CLIENT_CONFIGURATION".Namespaces.NamespaceCount, NodeIDCount := "DB16107_U03_MEAS_STA_MEAS_B_CLIENT_CONFIGURATION".ReadLists.U03_FACE_B_MEAS_Read.NodeCount, NamespaceUris := "DB16107_U03_MEAS_STA_MEAS_B_CLIENT_CONFIGURATION".Namespaces.NamespaceURIs, NamespaceStatusList := "DB16107_U03_MEAS_STA_MEAS_B_CLIENT_CONFIGURATION".Namespaces.NamespaceStatusList, NamespaceIndexes := "DB16107_U03_MEAS_STA_MEAS_B_CLIENT_CONFIGURATION".Namespaces.ServerNamespaceIndexes, NodeIDs := "DB16107_U03_MEAS_STA_MEAS_B_CLIENT_CONFIGURATION".ReadLists.U03_FACE_B_MEAS_Read.Nodes, NodeHdls := "DB16107_U03_MEAS_STA_MEAS_B_CLIENT_CONFIGURATION".ReadLists.U03_FACE_B_MEAS_Read.NodeHdls, NodeStatusList := "DB16007_U03_MEAS_STA_MEAS_B_CLIENT_INTERFACE".U03_FACE_B_MEAS_Read.NodeStatusList, Timestamps := "DB16007_U03_MEAS_STA_MEAS_B_CLIENT_INTERFACE".U03_FACE_B_MEAS_Read.TimeStamps, Variable := "DB16007_U03_MEAS_STA_MEAS_B_CLIENT_INTERFACE".U03_FACE_B_MEAS_Read.Variable, Done =>, Busy =>, Error =>, Status =>)
   END_RUNG
   // the same network as SCL:
   "DB16260_READLIST_U03_MEAS_B"(REQ := "DB16000_OPC_UA_TRIGGER_ALARM".CLIENT.U03_MEAS_STA_MEAS_B.TRIGGERS.READ_VARS,   // OPC_UA_ReadList_C
                           MaintainSession := true,
                           ServerEndpointUrl := "DB16107_U03_MEAS_STA_MEAS_B_CLIENT_CONFIGURATION".Connection.ServerEndpointUrl,
                           SessionConnectInfo := "DB16107_U03_MEAS_STA_MEAS_B_CLIENT_CONFIGURATION".Connection.ConnectInfo,
                           NamespaceUrisCount := "DB16107_U03_MEAS_STA_MEAS_B_CLIENT_CONFIGURATION".Namespaces.NamespaceCount,
                           NodeIDCount := "DB16107_U03_MEAS_STA_MEAS_B_CLIENT_CONFIGURATION".ReadLists.U03_FACE_B_MEAS_Read.NodeCount,
                           NamespaceUris := "DB16107_U03_MEAS_STA_MEAS_B_CLIENT_CONFIGURATION".Namespaces.NamespaceURIs,
                           NamespaceStatusList := "DB16107_U03_MEAS_STA_MEAS_B_CLIENT_CONFIGURATION".Namespaces.NamespaceStatusList,
                           NamespaceIndexes := "DB16107_U03_MEAS_STA_MEAS_B_CLIENT_CONFIGURATION".Namespaces.ServerNamespaceIndexes,
                           NodeIDs := "DB16107_U03_MEAS_STA_MEAS_B_CLIENT_CONFIGURATION".ReadLists.U03_FACE_B_MEAS_Read.Nodes,
                           NodeHdls := "DB16107_U03_MEAS_STA_MEAS_B_CLIENT_CONFIGURATION".ReadLists.U03_FACE_B_MEAS_Read.NodeHdls,
                           NodeStatusList := "DB16007_U03_MEAS_STA_MEAS_B_CLIENT_INTERFACE".U03_FACE_B_MEAS_Read.NodeStatusList,
                           Timestamps := "DB16007_U03_MEAS_STA_MEAS_B_CLIENT_INTERFACE".U03_FACE_B_MEAS_Read.TimeStamps,
                           Variable := "DB16007_U03_MEAS_STA_MEAS_B_CLIENT_INTERFACE".U03_FACE_B_MEAS_Read.Variable);
END_REGION

REGION Network 13: UNIT 03 FIXTURES CALIBRATION STATUS UPDATE
   RUNG wire#powerrail
      Contact( "M_ONE" )
      Contact( "DB16007_U03_MEAS_STA_MEAS_B_CLIENT_INTERFACE".U03_FACE_B_MEAS_Read.Variable."Status Fixture 1" )
      wire#w1
      Move(in := 1, out1 => "DB16010_MEASURE_SENSORS_CALIBRATION_STATUS".U03_STA_MEAS_MEAS_N.FIXTURE_1_STATUS)
   END_RUNG
   RUNG wire#w1
      Not()
      Move(in := 0, out1 => "DB16010_MEASURE_SENSORS_CALIBRATION_STATUS".U03_STA_MEAS_MEAS_N.FIXTURE_1_STATUS)
   END_RUNG
   // the same network as SCL:
   #_w1 := "M_ONE" AND "DB16007_U03_MEAS_STA_MEAS_B_CLIENT_INTERFACE".U03_FACE_B_MEAS_Read.Variable."Status Fixture 1";
   IF #_w1 THEN
       "DB16010_MEASURE_SENSORS_CALIBRATION_STATUS".U03_STA_MEAS_MEAS_N.FIXTURE_1_STATUS := 1;
   END_IF;
   IF NOT #_w1 THEN
       "DB16010_MEASURE_SENSORS_CALIBRATION_STATUS".U03_STA_MEAS_MEAS_N.FIXTURE_1_STATUS := 0;
   END_IF;
END_REGION

REGION Network 14: UNIT 03 MEASURING STATION FACE B MEASURING METHOD CONNECTION ALARM
   RUNG wire#powerrail
      Contact( "DB16261_METHODCALL_U03_MEAS_B_MEAS_TRIGGER".Error )
      wire#w1
      Contact( "DB7259_UNIT_03_STA_MEAS_B_ENABLE_DISABLE".ENABLED )
      wire#w2
      Coil( "DB16000_OPC_UA_TRIGGER_ALARM".CLIENT.U03_MEAS_STA_MEAS_B.ALARMS.MEAS_CONNECTION_A )
   END_RUNG
   RUNG wire#powerrail
      Contact( "DB16000_OPC_UA_TRIGGER_ALARM".CLIENT.U03_MEAS_STA_MEAS_B.ALARMS.MEAS_CONNECTION_A )
      I_Contact( "DB2120_MPP_ITC_IPC".RESET_FAULTS )
      I_Contact( "DB7300_INTERLOCK_GENERAL".GENERAL_MACHINE.FROM_CELL_TO_MACHINE_GENERAL.CELL_MEAS_STA_RESET )
   END_RUNG wire#w1
   RUNG wire#w2
      Coil( "DB426_ALARMS_WARNINGS".UNIT_03."724640" )
   END_RUNG
   // the same network as SCL:
   "DB16000_OPC_UA_TRIGGER_ALARM".CLIENT.U03_MEAS_STA_MEAS_B.ALARMS.MEAS_CONNECTION_A := ("DB16261_METHODCALL_U03_MEAS_B_MEAS_TRIGGER".Error OR ("DB16000_OPC_UA_TRIGGER_ALARM".CLIENT.U03_MEAS_STA_MEAS_B.ALARMS.MEAS_CONNECTION_A AND NOT "DB2120_MPP_ITC_IPC".RESET_FAULTS AND NOT "DB7300_INTERLOCK_GENERAL".GENERAL_MACHINE.FROM_CELL_TO_MACHINE_GENERAL.CELL_MEAS_STA_RESET)) AND "DB7259_UNIT_03_STA_MEAS_B_ENABLE_DISABLE".ENABLED;
   "DB426_ALARMS_WARNINGS".UNIT_03."724640" := "DB16000_OPC_UA_TRIGGER_ALARM".CLIENT.U03_MEAS_STA_MEAS_B.ALARMS.MEAS_CONNECTION_A;
END_REGION

REGION Network 15: UNIT 03 MEASURING STATION FACE B MEASURING METHOD WORKING OR BLOCKED ALARM
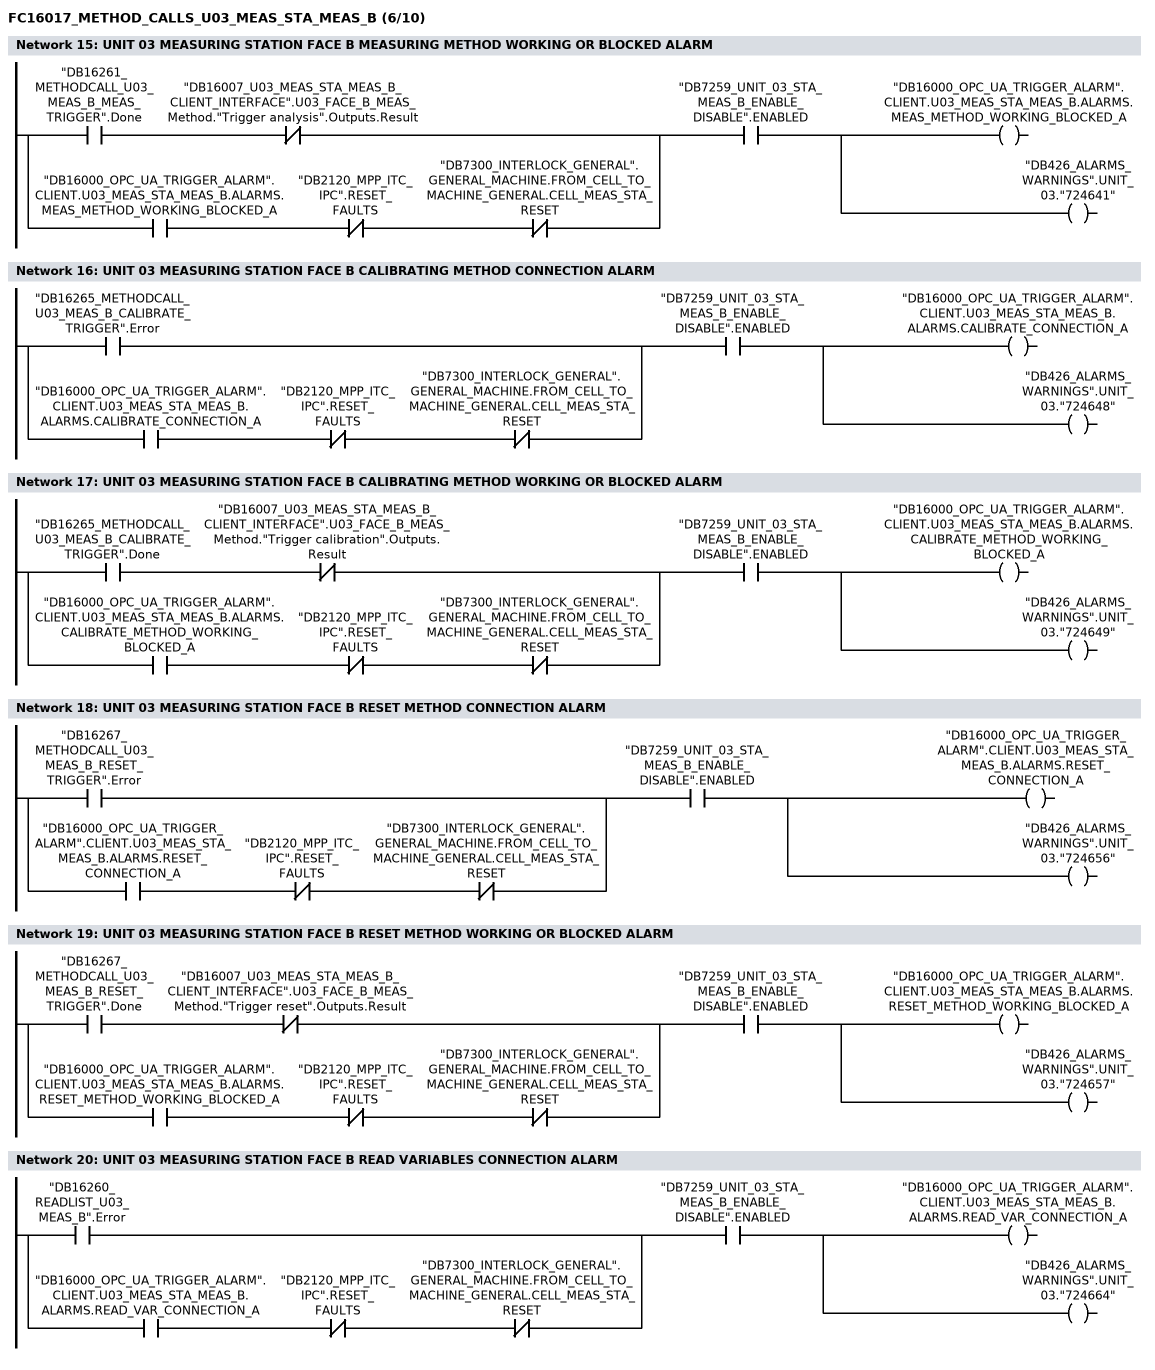
   RUNG wire#powerrail
      Contact( "DB16261_METHODCALL_U03_MEAS_B_MEAS_TRIGGER".Done )
      I_Contact( "DB16007_U03_MEAS_STA_MEAS_B_CLIENT_INTERFACE".U03_FACE_B_MEAS_Method."Trigger analysis".Outputs.Result )
      wire#w1
      Contact( "DB7259_UNIT_03_STA_MEAS_B_ENABLE_DISABLE".ENABLED )
      wire#w2
      Coil( "DB16000_OPC_UA_TRIGGER_ALARM".CLIENT.U03_MEAS_STA_MEAS_B.ALARMS.MEAS_METHOD_WORKING_BLOCKED_A )
   END_RUNG
   RUNG wire#powerrail
      Contact( "DB16000_OPC_UA_TRIGGER_ALARM".CLIENT.U03_MEAS_STA_MEAS_B.ALARMS.MEAS_METHOD_WORKING_BLOCKED_A )
      I_Contact( "DB2120_MPP_ITC_IPC".RESET_FAULTS )
      I_Contact( "DB7300_INTERLOCK_GENERAL".GENERAL_MACHINE.FROM_CELL_TO_MACHINE_GENERAL.CELL_MEAS_STA_RESET )
   END_RUNG wire#w1
   RUNG wire#w2
      Coil( "DB426_ALARMS_WARNINGS".UNIT_03."724641" )
   END_RUNG
   // the same network as SCL:
   "DB16000_OPC_UA_TRIGGER_ALARM".CLIENT.U03_MEAS_STA_MEAS_B.ALARMS.MEAS_METHOD_WORKING_BLOCKED_A := (("DB16261_METHODCALL_U03_MEAS_B_MEAS_TRIGGER".Done AND NOT "DB16007_U03_MEAS_STA_MEAS_B_CLIENT_INTERFACE".U03_FACE_B_MEAS_Method."Trigger analysis".Outputs.Result) OR ("DB16000_OPC_UA_TRIGGER_ALARM".CLIENT.U03_MEAS_STA_MEAS_B.ALARMS.MEAS_METHOD_WORKING_BLOCKED_A AND NOT "DB2120_MPP_ITC_IPC".RESET_FAULTS AND NOT "DB7300_INTERLOCK_GENERAL".GENERAL_MACHINE.FROM_CELL_TO_MACHINE_GENERAL.CELL_MEAS_STA_RESET)) AND "DB7259_UNIT_03_STA_MEAS_B_ENABLE_DISABLE".ENABLED;
   "DB426_ALARMS_WARNINGS".UNIT_03."724641" := "DB16000_OPC_UA_TRIGGER_ALARM".CLIENT.U03_MEAS_STA_MEAS_B.ALARMS.MEAS_METHOD_WORKING_BLOCKED_A;
END_REGION

REGION Network 16: UNIT 03 MEASURING STATION FACE B CALIBRATING METHOD CONNECTION ALARM
   RUNG wire#powerrail
      Contact( "DB16265_METHODCALL_U03_MEAS_B_CALIBRATE_TRIGGER".Error )
      wire#w1
      Contact( "DB7259_UNIT_03_STA_MEAS_B_ENABLE_DISABLE".ENABLED )
      wire#w2
      Coil( "DB16000_OPC_UA_TRIGGER_ALARM".CLIENT.U03_MEAS_STA_MEAS_B.ALARMS.CALIBRATE_CONNECTION_A )
   END_RUNG
   RUNG wire#powerrail
      Contact( "DB16000_OPC_UA_TRIGGER_ALARM".CLIENT.U03_MEAS_STA_MEAS_B.ALARMS.CALIBRATE_CONNECTION_A )
      I_Contact( "DB2120_MPP_ITC_IPC".RESET_FAULTS )
      I_Contact( "DB7300_INTERLOCK_GENERAL".GENERAL_MACHINE.FROM_CELL_TO_MACHINE_GENERAL.CELL_MEAS_STA_RESET )
   END_RUNG wire#w1
   RUNG wire#w2
      Coil( "DB426_ALARMS_WARNINGS".UNIT_03."724648" )
   END_RUNG
   // the same network as SCL:
   "DB16000_OPC_UA_TRIGGER_ALARM".CLIENT.U03_MEAS_STA_MEAS_B.ALARMS.CALIBRATE_CONNECTION_A := ("DB16265_METHODCALL_U03_MEAS_B_CALIBRATE_TRIGGER".Error OR ("DB16000_OPC_UA_TRIGGER_ALARM".CLIENT.U03_MEAS_STA_MEAS_B.ALARMS.CALIBRATE_CONNECTION_A AND NOT "DB2120_MPP_ITC_IPC".RESET_FAULTS AND NOT "DB7300_INTERLOCK_GENERAL".GENERAL_MACHINE.FROM_CELL_TO_MACHINE_GENERAL.CELL_MEAS_STA_RESET)) AND "DB7259_UNIT_03_STA_MEAS_B_ENABLE_DISABLE".ENABLED;
   "DB426_ALARMS_WARNINGS".UNIT_03."724648" := "DB16000_OPC_UA_TRIGGER_ALARM".CLIENT.U03_MEAS_STA_MEAS_B.ALARMS.CALIBRATE_CONNECTION_A;
END_REGION

REGION Network 17: UNIT 03 MEASURING STATION FACE B CALIBRATING METHOD WORKING OR BLOCKED ALARM
   RUNG wire#powerrail
      Contact( "DB16265_METHODCALL_U03_MEAS_B_CALIBRATE_TRIGGER".Done )
      I_Contact( "DB16007_U03_MEAS_STA_MEAS_B_CLIENT_INTERFACE".U03_FACE_B_MEAS_Method."Trigger calibration".Outputs.Result )
      wire#w1
      Contact( "DB7259_UNIT_03_STA_MEAS_B_ENABLE_DISABLE".ENABLED )
      wire#w2
      Coil( "DB16000_OPC_UA_TRIGGER_ALARM".CLIENT.U03_MEAS_STA_MEAS_B.ALARMS.CALIBRATE_METHOD_WORKING_BLOCKED_A )
   END_RUNG
   RUNG wire#powerrail
      Contact( "DB16000_OPC_UA_TRIGGER_ALARM".CLIENT.U03_MEAS_STA_MEAS_B.ALARMS.CALIBRATE_METHOD_WORKING_BLOCKED_A )
      I_Contact( "DB2120_MPP_ITC_IPC".RESET_FAULTS )
      I_Contact( "DB7300_INTERLOCK_GENERAL".GENERAL_MACHINE.FROM_CELL_TO_MACHINE_GENERAL.CELL_MEAS_STA_RESET )
   END_RUNG wire#w1
   RUNG wire#w2
      Coil( "DB426_ALARMS_WARNINGS".UNIT_03."724649" )
   END_RUNG
   // the same network as SCL:
   "DB16000_OPC_UA_TRIGGER_ALARM".CLIENT.U03_MEAS_STA_MEAS_B.ALARMS.CALIBRATE_METHOD_WORKING_BLOCKED_A := (("DB16265_METHODCALL_U03_MEAS_B_CALIBRATE_TRIGGER".Done AND NOT "DB16007_U03_MEAS_STA_MEAS_B_CLIENT_INTERFACE".U03_FACE_B_MEAS_Method."Trigger calibration".Outputs.Result) OR ("DB16000_OPC_UA_TRIGGER_ALARM".CLIENT.U03_MEAS_STA_MEAS_B.ALARMS.CALIBRATE_METHOD_WORKING_BLOCKED_A AND NOT "DB2120_MPP_ITC_IPC".RESET_FAULTS AND NOT "DB7300_INTERLOCK_GENERAL".GENERAL_MACHINE.FROM_CELL_TO_MACHINE_GENERAL.CELL_MEAS_STA_RESET)) AND "DB7259_UNIT_03_STA_MEAS_B_ENABLE_DISABLE".ENABLED;
   "DB426_ALARMS_WARNINGS".UNIT_03."724649" := "DB16000_OPC_UA_TRIGGER_ALARM".CLIENT.U03_MEAS_STA_MEAS_B.ALARMS.CALIBRATE_METHOD_WORKING_BLOCKED_A;
END_REGION

REGION Network 18: UNIT 03 MEASURING STATION FACE B RESET METHOD CONNECTION ALARM
   RUNG wire#powerrail
      Contact( "DB16267_METHODCALL_U03_MEAS_B_RESET_TRIGGER".Error )
      wire#w1
      Contact( "DB7259_UNIT_03_STA_MEAS_B_ENABLE_DISABLE".ENABLED )
      wire#w2
      Coil( "DB16000_OPC_UA_TRIGGER_ALARM".CLIENT.U03_MEAS_STA_MEAS_B.ALARMS.RESET_CONNECTION_A )
   END_RUNG
   RUNG wire#powerrail
      Contact( "DB16000_OPC_UA_TRIGGER_ALARM".CLIENT.U03_MEAS_STA_MEAS_B.ALARMS.RESET_CONNECTION_A )
      I_Contact( "DB2120_MPP_ITC_IPC".RESET_FAULTS )
      I_Contact( "DB7300_INTERLOCK_GENERAL".GENERAL_MACHINE.FROM_CELL_TO_MACHINE_GENERAL.CELL_MEAS_STA_RESET )
   END_RUNG wire#w1
   RUNG wire#w2
      Coil( "DB426_ALARMS_WARNINGS".UNIT_03."724656" )
   END_RUNG
   // the same network as SCL:
   "DB16000_OPC_UA_TRIGGER_ALARM".CLIENT.U03_MEAS_STA_MEAS_B.ALARMS.RESET_CONNECTION_A := ("DB16267_METHODCALL_U03_MEAS_B_RESET_TRIGGER".Error OR ("DB16000_OPC_UA_TRIGGER_ALARM".CLIENT.U03_MEAS_STA_MEAS_B.ALARMS.RESET_CONNECTION_A AND NOT "DB2120_MPP_ITC_IPC".RESET_FAULTS AND NOT "DB7300_INTERLOCK_GENERAL".GENERAL_MACHINE.FROM_CELL_TO_MACHINE_GENERAL.CELL_MEAS_STA_RESET)) AND "DB7259_UNIT_03_STA_MEAS_B_ENABLE_DISABLE".ENABLED;
   "DB426_ALARMS_WARNINGS".UNIT_03."724656" := "DB16000_OPC_UA_TRIGGER_ALARM".CLIENT.U03_MEAS_STA_MEAS_B.ALARMS.RESET_CONNECTION_A;
END_REGION

REGION Network 19: UNIT 03 MEASURING STATION FACE B RESET METHOD WORKING OR BLOCKED ALARM
   RUNG wire#powerrail
      Contact( "DB16267_METHODCALL_U03_MEAS_B_RESET_TRIGGER".Done )
      I_Contact( "DB16007_U03_MEAS_STA_MEAS_B_CLIENT_INTERFACE".U03_FACE_B_MEAS_Method."Trigger reset".Outputs.Result )
      wire#w1
      Contact( "DB7259_UNIT_03_STA_MEAS_B_ENABLE_DISABLE".ENABLED )
      wire#w2
      Coil( "DB16000_OPC_UA_TRIGGER_ALARM".CLIENT.U03_MEAS_STA_MEAS_B.ALARMS.RESET_METHOD_WORKING_BLOCKED_A )
   END_RUNG
   RUNG wire#powerrail
      Contact( "DB16000_OPC_UA_TRIGGER_ALARM".CLIENT.U03_MEAS_STA_MEAS_B.ALARMS.RESET_METHOD_WORKING_BLOCKED_A )
      I_Contact( "DB2120_MPP_ITC_IPC".RESET_FAULTS )
      I_Contact( "DB7300_INTERLOCK_GENERAL".GENERAL_MACHINE.FROM_CELL_TO_MACHINE_GENERAL.CELL_MEAS_STA_RESET )
   END_RUNG wire#w1
   RUNG wire#w2
      Coil( "DB426_ALARMS_WARNINGS".UNIT_03."724657" )
   END_RUNG
   // the same network as SCL:
   "DB16000_OPC_UA_TRIGGER_ALARM".CLIENT.U03_MEAS_STA_MEAS_B.ALARMS.RESET_METHOD_WORKING_BLOCKED_A := (("DB16267_METHODCALL_U03_MEAS_B_RESET_TRIGGER".Done AND NOT "DB16007_U03_MEAS_STA_MEAS_B_CLIENT_INTERFACE".U03_FACE_B_MEAS_Method."Trigger reset".Outputs.Result) OR ("DB16000_OPC_UA_TRIGGER_ALARM".CLIENT.U03_MEAS_STA_MEAS_B.ALARMS.RESET_METHOD_WORKING_BLOCKED_A AND NOT "DB2120_MPP_ITC_IPC".RESET_FAULTS AND NOT "DB7300_INTERLOCK_GENERAL".GENERAL_MACHINE.FROM_CELL_TO_MACHINE_GENERAL.CELL_MEAS_STA_RESET)) AND "DB7259_UNIT_03_STA_MEAS_B_ENABLE_DISABLE".ENABLED;
   "DB426_ALARMS_WARNINGS".UNIT_03."724657" := "DB16000_OPC_UA_TRIGGER_ALARM".CLIENT.U03_MEAS_STA_MEAS_B.ALARMS.RESET_METHOD_WORKING_BLOCKED_A;
END_REGION

REGION Network 20: UNIT 03 MEASURING STATION FACE B READ VARIABLES CONNECTION ALARM
   RUNG wire#powerrail
      Contact( "DB16260_READLIST_U03_MEAS_B".Error )
      wire#w1
      Contact( "DB7259_UNIT_03_STA_MEAS_B_ENABLE_DISABLE".ENABLED )
      wire#w2
      Coil( "DB16000_OPC_UA_TRIGGER_ALARM".CLIENT.U03_MEAS_STA_MEAS_B.ALARMS.READ_VAR_CONNECTION_A )
   END_RUNG
   RUNG wire#powerrail
      Contact( "DB16000_OPC_UA_TRIGGER_ALARM".CLIENT.U03_MEAS_STA_MEAS_B.ALARMS.READ_VAR_CONNECTION_A )
      I_Contact( "DB2120_MPP_ITC_IPC".RESET_FAULTS )
      I_Contact( "DB7300_INTERLOCK_GENERAL".GENERAL_MACHINE.FROM_CELL_TO_MACHINE_GENERAL.CELL_MEAS_STA_RESET )
   END_RUNG wire#w1
   RUNG wire#w2
      Coil( "DB426_ALARMS_WARNINGS".UNIT_03."724664" )
   END_RUNG
   // the same network as SCL:
   "DB16000_OPC_UA_TRIGGER_ALARM".CLIENT.U03_MEAS_STA_MEAS_B.ALARMS.READ_VAR_CONNECTION_A := ("DB16260_READLIST_U03_MEAS_B".Error OR ("DB16000_OPC_UA_TRIGGER_ALARM".CLIENT.U03_MEAS_STA_MEAS_B.ALARMS.READ_VAR_CONNECTION_A AND NOT "DB2120_MPP_ITC_IPC".RESET_FAULTS AND NOT "DB7300_INTERLOCK_GENERAL".GENERAL_MACHINE.FROM_CELL_TO_MACHINE_GENERAL.CELL_MEAS_STA_RESET)) AND "DB7259_UNIT_03_STA_MEAS_B_ENABLE_DISABLE".ENABLED;
   "DB426_ALARMS_WARNINGS".UNIT_03."724664" := "DB16000_OPC_UA_TRIGGER_ALARM".CLIENT.U03_MEAS_STA_MEAS_B.ALARMS.READ_VAR_CONNECTION_A;
END_REGION

REGION Network 21: UNIT 03 MEASURING STATION FACE B READ VARIABLES WORKING OR BLOCKED ALARM
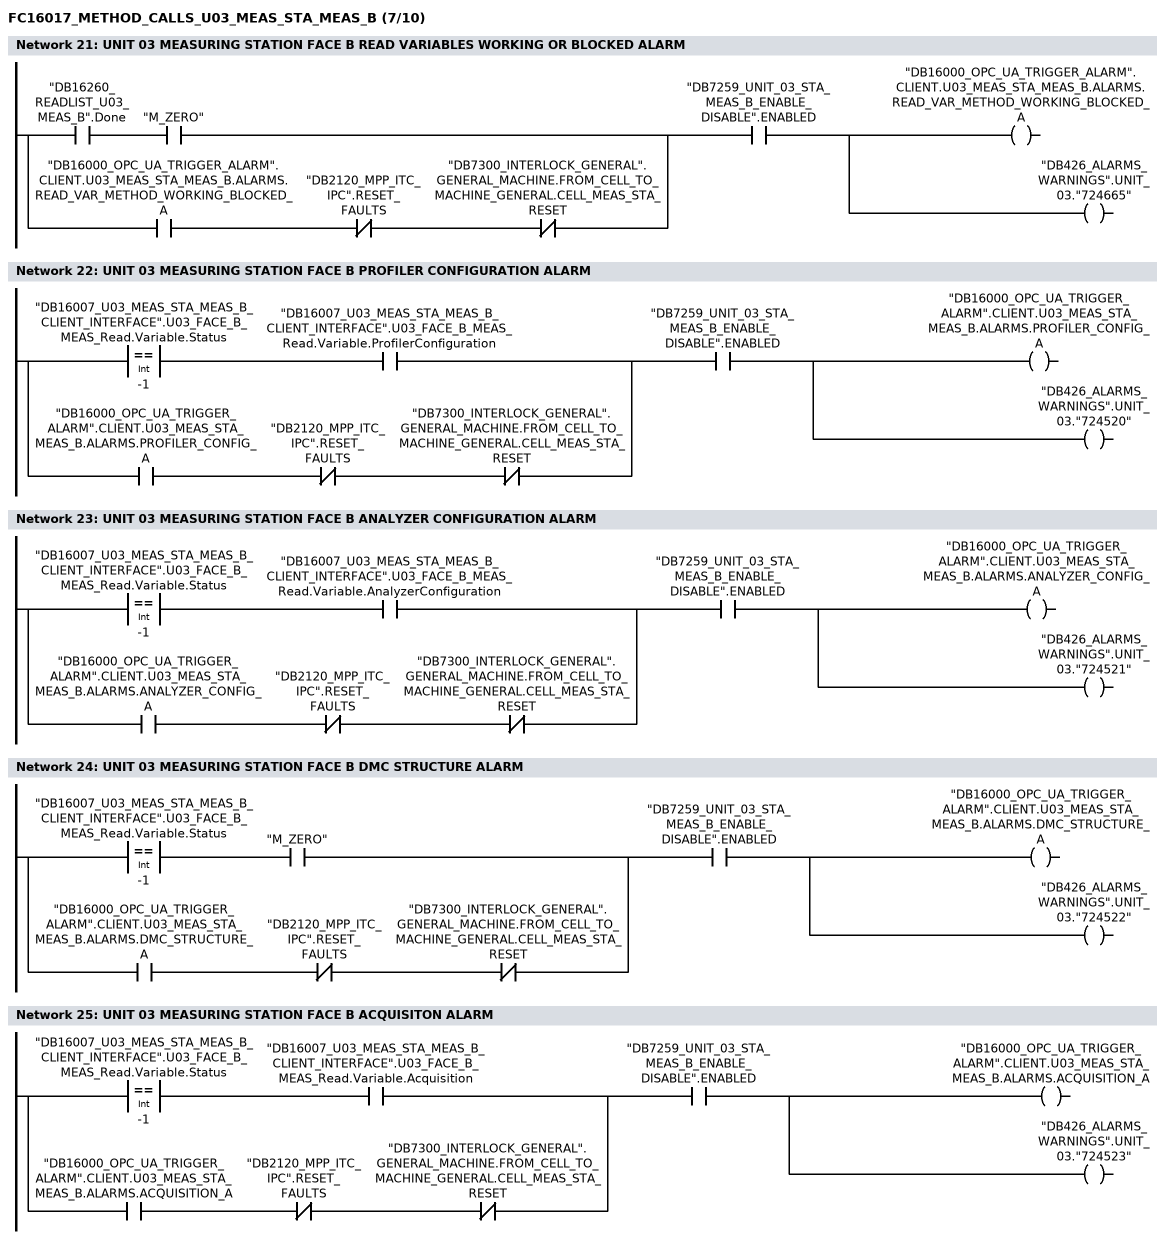
   RUNG wire#powerrail
      Contact( "DB16260_READLIST_U03_MEAS_B".Done )
      Contact( "M_ZERO" )
      wire#w1
      Contact( "DB7259_UNIT_03_STA_MEAS_B_ENABLE_DISABLE".ENABLED )
      wire#w2
      Coil( "DB16000_OPC_UA_TRIGGER_ALARM".CLIENT.U03_MEAS_STA_MEAS_B.ALARMS.READ_VAR_METHOD_WORKING_BLOCKED_A )
   END_RUNG
   RUNG wire#powerrail
      Contact( "DB16000_OPC_UA_TRIGGER_ALARM".CLIENT.U03_MEAS_STA_MEAS_B.ALARMS.READ_VAR_METHOD_WORKING_BLOCKED_A )
      I_Contact( "DB2120_MPP_ITC_IPC".RESET_FAULTS )
      I_Contact( "DB7300_INTERLOCK_GENERAL".GENERAL_MACHINE.FROM_CELL_TO_MACHINE_GENERAL.CELL_MEAS_STA_RESET )
   END_RUNG wire#w1
   RUNG wire#w2
      Coil( "DB426_ALARMS_WARNINGS".UNIT_03."724665" )
   END_RUNG
   // the same network as SCL:
   "DB16000_OPC_UA_TRIGGER_ALARM".CLIENT.U03_MEAS_STA_MEAS_B.ALARMS.READ_VAR_METHOD_WORKING_BLOCKED_A := (("DB16260_READLIST_U03_MEAS_B".Done AND "M_ZERO") OR ("DB16000_OPC_UA_TRIGGER_ALARM".CLIENT.U03_MEAS_STA_MEAS_B.ALARMS.READ_VAR_METHOD_WORKING_BLOCKED_A AND NOT "DB2120_MPP_ITC_IPC".RESET_FAULTS AND NOT "DB7300_INTERLOCK_GENERAL".GENERAL_MACHINE.FROM_CELL_TO_MACHINE_GENERAL.CELL_MEAS_STA_RESET)) AND "DB7259_UNIT_03_STA_MEAS_B_ENABLE_DISABLE".ENABLED;
   "DB426_ALARMS_WARNINGS".UNIT_03."724665" := "DB16000_OPC_UA_TRIGGER_ALARM".CLIENT.U03_MEAS_STA_MEAS_B.ALARMS.READ_VAR_METHOD_WORKING_BLOCKED_A;
END_REGION

REGION Network 22: UNIT 03 MEASURING STATION FACE B PROFILER CONFIGURATION ALARM
   RUNG wire#powerrail
      { S7_Templates := "SrcType := Int" } EQ_Contact(in1 := "DB16007_U03_MEAS_STA_MEAS_B_CLIENT_INTERFACE".U03_FACE_B_MEAS_Read.Variable.Status, in2 := -1)
      Contact( "DB16007_U03_MEAS_STA_MEAS_B_CLIENT_INTERFACE".U03_FACE_B_MEAS_Read.Variable.ProfilerConfiguration )
      wire#w1
      Contact( "DB7259_UNIT_03_STA_MEAS_B_ENABLE_DISABLE".ENABLED )
      wire#w2
      Coil( "DB16000_OPC_UA_TRIGGER_ALARM".CLIENT.U03_MEAS_STA_MEAS_B.ALARMS.PROFILER_CONFIG_A )
   END_RUNG
   RUNG wire#powerrail
      Contact( "DB16000_OPC_UA_TRIGGER_ALARM".CLIENT.U03_MEAS_STA_MEAS_B.ALARMS.PROFILER_CONFIG_A )
      I_Contact( "DB2120_MPP_ITC_IPC".RESET_FAULTS )
      I_Contact( "DB7300_INTERLOCK_GENERAL".GENERAL_MACHINE.FROM_CELL_TO_MACHINE_GENERAL.CELL_MEAS_STA_RESET )
   END_RUNG wire#w1
   RUNG wire#w2
      Coil( "DB426_ALARMS_WARNINGS".UNIT_03."724520" )
   END_RUNG
   // the same network as SCL:
   "DB16000_OPC_UA_TRIGGER_ALARM".CLIENT.U03_MEAS_STA_MEAS_B.ALARMS.PROFILER_CONFIG_A := ((("DB16007_U03_MEAS_STA_MEAS_B_CLIENT_INTERFACE".U03_FACE_B_MEAS_Read.Variable.Status = (-1)) AND "DB16007_U03_MEAS_STA_MEAS_B_CLIENT_INTERFACE".U03_FACE_B_MEAS_Read.Variable.ProfilerConfiguration) OR ("DB16000_OPC_UA_TRIGGER_ALARM".CLIENT.U03_MEAS_STA_MEAS_B.ALARMS.PROFILER_CONFIG_A AND NOT "DB2120_MPP_ITC_IPC".RESET_FAULTS AND NOT "DB7300_INTERLOCK_GENERAL".GENERAL_MACHINE.FROM_CELL_TO_MACHINE_GENERAL.CELL_MEAS_STA_RESET)) AND "DB7259_UNIT_03_STA_MEAS_B_ENABLE_DISABLE".ENABLED;
   "DB426_ALARMS_WARNINGS".UNIT_03."724520" := "DB16000_OPC_UA_TRIGGER_ALARM".CLIENT.U03_MEAS_STA_MEAS_B.ALARMS.PROFILER_CONFIG_A;
END_REGION

REGION Network 23: UNIT 03 MEASURING STATION FACE B ANALYZER CONFIGURATION ALARM
   RUNG wire#powerrail
      { S7_Templates := "SrcType := Int" } EQ_Contact(in1 := "DB16007_U03_MEAS_STA_MEAS_B_CLIENT_INTERFACE".U03_FACE_B_MEAS_Read.Variable.Status, in2 := -1)
      Contact( "DB16007_U03_MEAS_STA_MEAS_B_CLIENT_INTERFACE".U03_FACE_B_MEAS_Read.Variable.AnalyzerConfiguration )
      wire#w1
      Contact( "DB7259_UNIT_03_STA_MEAS_B_ENABLE_DISABLE".ENABLED )
      wire#w2
      Coil( "DB16000_OPC_UA_TRIGGER_ALARM".CLIENT.U03_MEAS_STA_MEAS_B.ALARMS.ANALYZER_CONFIG_A )
   END_RUNG
   RUNG wire#powerrail
      Contact( "DB16000_OPC_UA_TRIGGER_ALARM".CLIENT.U03_MEAS_STA_MEAS_B.ALARMS.ANALYZER_CONFIG_A )
      I_Contact( "DB2120_MPP_ITC_IPC".RESET_FAULTS )
      I_Contact( "DB7300_INTERLOCK_GENERAL".GENERAL_MACHINE.FROM_CELL_TO_MACHINE_GENERAL.CELL_MEAS_STA_RESET )
   END_RUNG wire#w1
   RUNG wire#w2
      Coil( "DB426_ALARMS_WARNINGS".UNIT_03."724521" )
   END_RUNG
   // the same network as SCL:
   "DB16000_OPC_UA_TRIGGER_ALARM".CLIENT.U03_MEAS_STA_MEAS_B.ALARMS.ANALYZER_CONFIG_A := ((("DB16007_U03_MEAS_STA_MEAS_B_CLIENT_INTERFACE".U03_FACE_B_MEAS_Read.Variable.Status = (-1)) AND "DB16007_U03_MEAS_STA_MEAS_B_CLIENT_INTERFACE".U03_FACE_B_MEAS_Read.Variable.AnalyzerConfiguration) OR ("DB16000_OPC_UA_TRIGGER_ALARM".CLIENT.U03_MEAS_STA_MEAS_B.ALARMS.ANALYZER_CONFIG_A AND NOT "DB2120_MPP_ITC_IPC".RESET_FAULTS AND NOT "DB7300_INTERLOCK_GENERAL".GENERAL_MACHINE.FROM_CELL_TO_MACHINE_GENERAL.CELL_MEAS_STA_RESET)) AND "DB7259_UNIT_03_STA_MEAS_B_ENABLE_DISABLE".ENABLED;
   "DB426_ALARMS_WARNINGS".UNIT_03."724521" := "DB16000_OPC_UA_TRIGGER_ALARM".CLIENT.U03_MEAS_STA_MEAS_B.ALARMS.ANALYZER_CONFIG_A;
END_REGION

REGION Network 24: UNIT 03 MEASURING STATION FACE B DMC STRUCTURE ALARM
   RUNG wire#powerrail
      { S7_Templates := "SrcType := Int" } EQ_Contact(in1 := "DB16007_U03_MEAS_STA_MEAS_B_CLIENT_INTERFACE".U03_FACE_B_MEAS_Read.Variable.Status, in2 := -1)
      Contact( "M_ZERO" )
      wire#w1
      Contact( "DB7259_UNIT_03_STA_MEAS_B_ENABLE_DISABLE".ENABLED )
      wire#w2
      Coil( "DB16000_OPC_UA_TRIGGER_ALARM".CLIENT.U03_MEAS_STA_MEAS_B.ALARMS.DMC_STRUCTURE_A )
   END_RUNG
   RUNG wire#powerrail
      Contact( "DB16000_OPC_UA_TRIGGER_ALARM".CLIENT.U03_MEAS_STA_MEAS_B.ALARMS.DMC_STRUCTURE_A )
      I_Contact( "DB2120_MPP_ITC_IPC".RESET_FAULTS )
      I_Contact( "DB7300_INTERLOCK_GENERAL".GENERAL_MACHINE.FROM_CELL_TO_MACHINE_GENERAL.CELL_MEAS_STA_RESET )
   END_RUNG wire#w1
   RUNG wire#w2
      Coil( "DB426_ALARMS_WARNINGS".UNIT_03."724522" )
   END_RUNG
   // the same network as SCL:
   "DB16000_OPC_UA_TRIGGER_ALARM".CLIENT.U03_MEAS_STA_MEAS_B.ALARMS.DMC_STRUCTURE_A := ((("DB16007_U03_MEAS_STA_MEAS_B_CLIENT_INTERFACE".U03_FACE_B_MEAS_Read.Variable.Status = (-1)) AND "M_ZERO") OR ("DB16000_OPC_UA_TRIGGER_ALARM".CLIENT.U03_MEAS_STA_MEAS_B.ALARMS.DMC_STRUCTURE_A AND NOT "DB2120_MPP_ITC_IPC".RESET_FAULTS AND NOT "DB7300_INTERLOCK_GENERAL".GENERAL_MACHINE.FROM_CELL_TO_MACHINE_GENERAL.CELL_MEAS_STA_RESET)) AND "DB7259_UNIT_03_STA_MEAS_B_ENABLE_DISABLE".ENABLED;
   "DB426_ALARMS_WARNINGS".UNIT_03."724522" := "DB16000_OPC_UA_TRIGGER_ALARM".CLIENT.U03_MEAS_STA_MEAS_B.ALARMS.DMC_STRUCTURE_A;
END_REGION

REGION Network 25: UNIT 03 MEASURING STATION FACE B ACQUISITON ALARM
   RUNG wire#powerrail
      { S7_Templates := "SrcType := Int" } EQ_Contact(in1 := "DB16007_U03_MEAS_STA_MEAS_B_CLIENT_INTERFACE".U03_FACE_B_MEAS_Read.Variable.Status, in2 := -1)
      Contact( "DB16007_U03_MEAS_STA_MEAS_B_CLIENT_INTERFACE".U03_FACE_B_MEAS_Read.Variable.Acquisition )
      wire#w1
      Contact( "DB7259_UNIT_03_STA_MEAS_B_ENABLE_DISABLE".ENABLED )
      wire#w2
      Coil( "DB16000_OPC_UA_TRIGGER_ALARM".CLIENT.U03_MEAS_STA_MEAS_B.ALARMS.ACQUISITION_A )
   END_RUNG
   RUNG wire#powerrail
      Contact( "DB16000_OPC_UA_TRIGGER_ALARM".CLIENT.U03_MEAS_STA_MEAS_B.ALARMS.ACQUISITION_A )
      I_Contact( "DB2120_MPP_ITC_IPC".RESET_FAULTS )
      I_Contact( "DB7300_INTERLOCK_GENERAL".GENERAL_MACHINE.FROM_CELL_TO_MACHINE_GENERAL.CELL_MEAS_STA_RESET )
   END_RUNG wire#w1
   RUNG wire#w2
      Coil( "DB426_ALARMS_WARNINGS".UNIT_03."724523" )
   END_RUNG
   // the same network as SCL:
   "DB16000_OPC_UA_TRIGGER_ALARM".CLIENT.U03_MEAS_STA_MEAS_B.ALARMS.ACQUISITION_A := ((("DB16007_U03_MEAS_STA_MEAS_B_CLIENT_INTERFACE".U03_FACE_B_MEAS_Read.Variable.Status = (-1)) AND "DB16007_U03_MEAS_STA_MEAS_B_CLIENT_INTERFACE".U03_FACE_B_MEAS_Read.Variable.Acquisition) OR ("DB16000_OPC_UA_TRIGGER_ALARM".CLIENT.U03_MEAS_STA_MEAS_B.ALARMS.ACQUISITION_A AND NOT "DB2120_MPP_ITC_IPC".RESET_FAULTS AND NOT "DB7300_INTERLOCK_GENERAL".GENERAL_MACHINE.FROM_CELL_TO_MACHINE_GENERAL.CELL_MEAS_STA_RESET)) AND "DB7259_UNIT_03_STA_MEAS_B_ENABLE_DISABLE".ENABLED;
   "DB426_ALARMS_WARNINGS".UNIT_03."724523" := "DB16000_OPC_UA_TRIGGER_ALARM".CLIENT.U03_MEAS_STA_MEAS_B.ALARMS.ACQUISITION_A;
END_REGION

REGION Network 26: UNIT 03 MEASURING STATION FACE B PROFILER INITIALIZTION ALARM
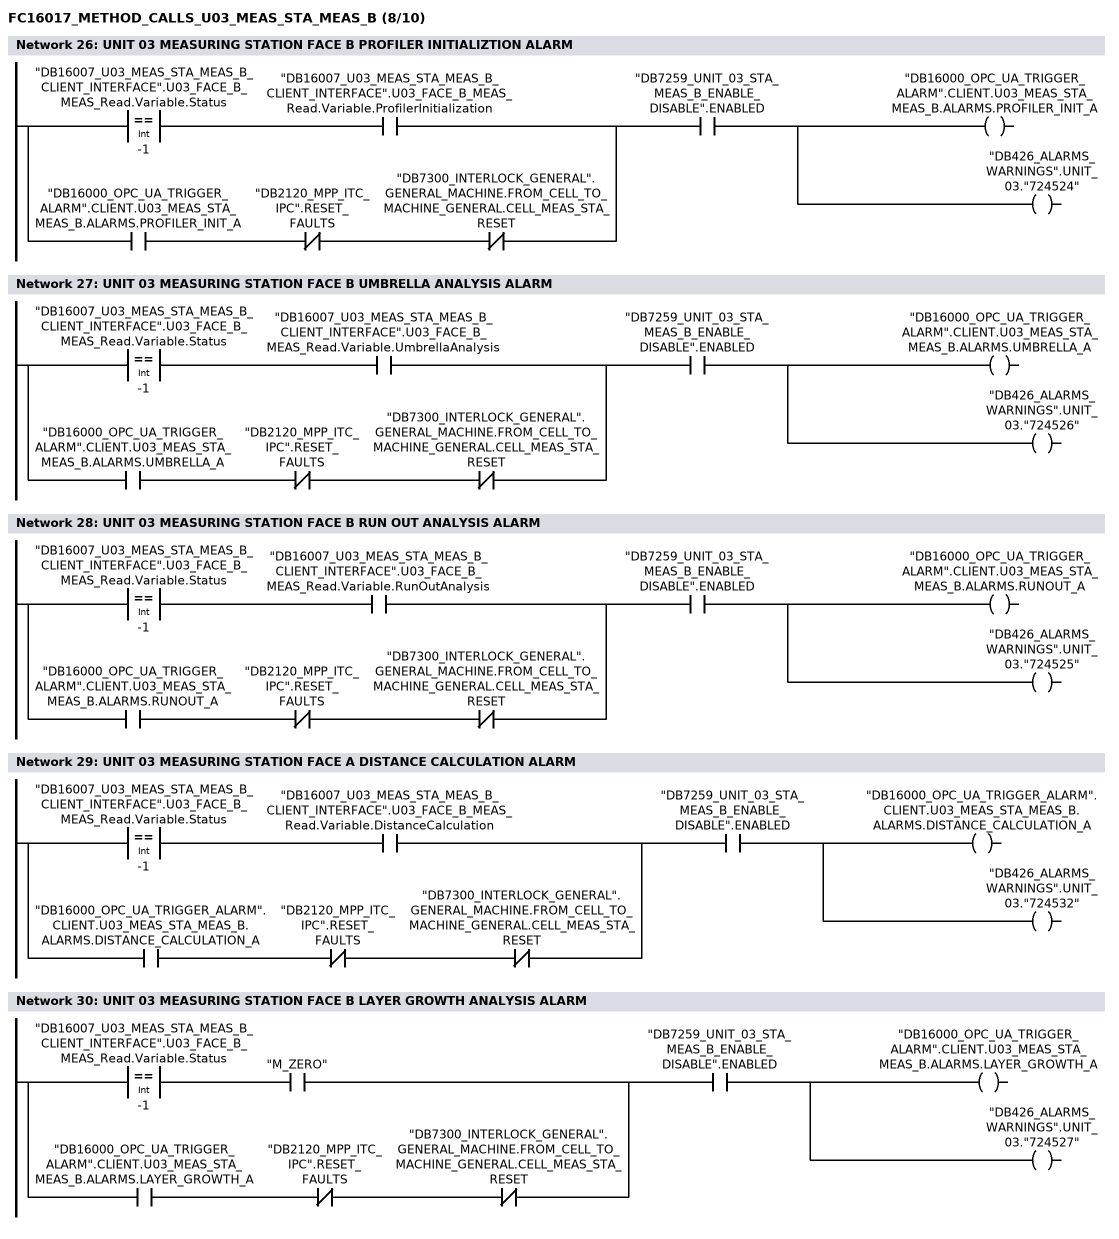
   RUNG wire#powerrail
      { S7_Templates := "SrcType := Int" } EQ_Contact(in1 := "DB16007_U03_MEAS_STA_MEAS_B_CLIENT_INTERFACE".U03_FACE_B_MEAS_Read.Variable.Status, in2 := -1)
      Contact( "DB16007_U03_MEAS_STA_MEAS_B_CLIENT_INTERFACE".U03_FACE_B_MEAS_Read.Variable.ProfilerInitialization )
      wire#w1
      Contact( "DB7259_UNIT_03_STA_MEAS_B_ENABLE_DISABLE".ENABLED )
      wire#w2
      Coil( "DB16000_OPC_UA_TRIGGER_ALARM".CLIENT.U03_MEAS_STA_MEAS_B.ALARMS.PROFILER_INIT_A )
   END_RUNG
   RUNG wire#powerrail
      Contact( "DB16000_OPC_UA_TRIGGER_ALARM".CLIENT.U03_MEAS_STA_MEAS_B.ALARMS.PROFILER_INIT_A )
      I_Contact( "DB2120_MPP_ITC_IPC".RESET_FAULTS )
      I_Contact( "DB7300_INTERLOCK_GENERAL".GENERAL_MACHINE.FROM_CELL_TO_MACHINE_GENERAL.CELL_MEAS_STA_RESET )
   END_RUNG wire#w1
   RUNG wire#w2
      Coil( "DB426_ALARMS_WARNINGS".UNIT_03."724524" )
   END_RUNG
   // the same network as SCL:
   "DB16000_OPC_UA_TRIGGER_ALARM".CLIENT.U03_MEAS_STA_MEAS_B.ALARMS.PROFILER_INIT_A := ((("DB16007_U03_MEAS_STA_MEAS_B_CLIENT_INTERFACE".U03_FACE_B_MEAS_Read.Variable.Status = (-1)) AND "DB16007_U03_MEAS_STA_MEAS_B_CLIENT_INTERFACE".U03_FACE_B_MEAS_Read.Variable.ProfilerInitialization) OR ("DB16000_OPC_UA_TRIGGER_ALARM".CLIENT.U03_MEAS_STA_MEAS_B.ALARMS.PROFILER_INIT_A AND NOT "DB2120_MPP_ITC_IPC".RESET_FAULTS AND NOT "DB7300_INTERLOCK_GENERAL".GENERAL_MACHINE.FROM_CELL_TO_MACHINE_GENERAL.CELL_MEAS_STA_RESET)) AND "DB7259_UNIT_03_STA_MEAS_B_ENABLE_DISABLE".ENABLED;
   "DB426_ALARMS_WARNINGS".UNIT_03."724524" := "DB16000_OPC_UA_TRIGGER_ALARM".CLIENT.U03_MEAS_STA_MEAS_B.ALARMS.PROFILER_INIT_A;
END_REGION

REGION Network 27: UNIT 03 MEASURING STATION FACE B UMBRELLA ANALYSIS ALARM
   RUNG wire#powerrail
      { S7_Templates := "SrcType := Int" } EQ_Contact(in1 := "DB16007_U03_MEAS_STA_MEAS_B_CLIENT_INTERFACE".U03_FACE_B_MEAS_Read.Variable.Status, in2 := -1)
      Contact( "DB16007_U03_MEAS_STA_MEAS_B_CLIENT_INTERFACE".U03_FACE_B_MEAS_Read.Variable.UmbrellaAnalysis )
      wire#w1
      Contact( "DB7259_UNIT_03_STA_MEAS_B_ENABLE_DISABLE".ENABLED )
      wire#w2
      Coil( "DB16000_OPC_UA_TRIGGER_ALARM".CLIENT.U03_MEAS_STA_MEAS_B.ALARMS.UMBRELLA_A )
   END_RUNG
   RUNG wire#powerrail
      Contact( "DB16000_OPC_UA_TRIGGER_ALARM".CLIENT.U03_MEAS_STA_MEAS_B.ALARMS.UMBRELLA_A )
      I_Contact( "DB2120_MPP_ITC_IPC".RESET_FAULTS )
      I_Contact( "DB7300_INTERLOCK_GENERAL".GENERAL_MACHINE.FROM_CELL_TO_MACHINE_GENERAL.CELL_MEAS_STA_RESET )
   END_RUNG wire#w1
   RUNG wire#w2
      Coil( "DB426_ALARMS_WARNINGS".UNIT_03."724526" )
   END_RUNG
   // the same network as SCL:
   "DB16000_OPC_UA_TRIGGER_ALARM".CLIENT.U03_MEAS_STA_MEAS_B.ALARMS.UMBRELLA_A := ((("DB16007_U03_MEAS_STA_MEAS_B_CLIENT_INTERFACE".U03_FACE_B_MEAS_Read.Variable.Status = (-1)) AND "DB16007_U03_MEAS_STA_MEAS_B_CLIENT_INTERFACE".U03_FACE_B_MEAS_Read.Variable.UmbrellaAnalysis) OR ("DB16000_OPC_UA_TRIGGER_ALARM".CLIENT.U03_MEAS_STA_MEAS_B.ALARMS.UMBRELLA_A AND NOT "DB2120_MPP_ITC_IPC".RESET_FAULTS AND NOT "DB7300_INTERLOCK_GENERAL".GENERAL_MACHINE.FROM_CELL_TO_MACHINE_GENERAL.CELL_MEAS_STA_RESET)) AND "DB7259_UNIT_03_STA_MEAS_B_ENABLE_DISABLE".ENABLED;
   "DB426_ALARMS_WARNINGS".UNIT_03."724526" := "DB16000_OPC_UA_TRIGGER_ALARM".CLIENT.U03_MEAS_STA_MEAS_B.ALARMS.UMBRELLA_A;
END_REGION

REGION Network 28: UNIT 03 MEASURING STATION FACE B RUN OUT ANALYSIS ALARM
   RUNG wire#powerrail
      { S7_Templates := "SrcType := Int" } EQ_Contact(in1 := "DB16007_U03_MEAS_STA_MEAS_B_CLIENT_INTERFACE".U03_FACE_B_MEAS_Read.Variable.Status, in2 := -1)
      Contact( "DB16007_U03_MEAS_STA_MEAS_B_CLIENT_INTERFACE".U03_FACE_B_MEAS_Read.Variable.RunOutAnalysis )
      wire#w1
      Contact( "DB7259_UNIT_03_STA_MEAS_B_ENABLE_DISABLE".ENABLED )
      wire#w2
      Coil( "DB16000_OPC_UA_TRIGGER_ALARM".CLIENT.U03_MEAS_STA_MEAS_B.ALARMS.RUNOUT_A )
   END_RUNG
   RUNG wire#powerrail
      Contact( "DB16000_OPC_UA_TRIGGER_ALARM".CLIENT.U03_MEAS_STA_MEAS_B.ALARMS.RUNOUT_A )
      I_Contact( "DB2120_MPP_ITC_IPC".RESET_FAULTS )
      I_Contact( "DB7300_INTERLOCK_GENERAL".GENERAL_MACHINE.FROM_CELL_TO_MACHINE_GENERAL.CELL_MEAS_STA_RESET )
   END_RUNG wire#w1
   RUNG wire#w2
      Coil( "DB426_ALARMS_WARNINGS".UNIT_03."724525" )
   END_RUNG
   // the same network as SCL:
   "DB16000_OPC_UA_TRIGGER_ALARM".CLIENT.U03_MEAS_STA_MEAS_B.ALARMS.RUNOUT_A := ((("DB16007_U03_MEAS_STA_MEAS_B_CLIENT_INTERFACE".U03_FACE_B_MEAS_Read.Variable.Status = (-1)) AND "DB16007_U03_MEAS_STA_MEAS_B_CLIENT_INTERFACE".U03_FACE_B_MEAS_Read.Variable.RunOutAnalysis) OR ("DB16000_OPC_UA_TRIGGER_ALARM".CLIENT.U03_MEAS_STA_MEAS_B.ALARMS.RUNOUT_A AND NOT "DB2120_MPP_ITC_IPC".RESET_FAULTS AND NOT "DB7300_INTERLOCK_GENERAL".GENERAL_MACHINE.FROM_CELL_TO_MACHINE_GENERAL.CELL_MEAS_STA_RESET)) AND "DB7259_UNIT_03_STA_MEAS_B_ENABLE_DISABLE".ENABLED;
   "DB426_ALARMS_WARNINGS".UNIT_03."724525" := "DB16000_OPC_UA_TRIGGER_ALARM".CLIENT.U03_MEAS_STA_MEAS_B.ALARMS.RUNOUT_A;
END_REGION

REGION Network 29: UNIT 03 MEASURING STATION FACE A DISTANCE CALCULATION ALARM
   RUNG wire#powerrail
      { S7_Templates := "SrcType := Int" } EQ_Contact(in1 := "DB16007_U03_MEAS_STA_MEAS_B_CLIENT_INTERFACE".U03_FACE_B_MEAS_Read.Variable.Status, in2 := -1)
      Contact( "DB16007_U03_MEAS_STA_MEAS_B_CLIENT_INTERFACE".U03_FACE_B_MEAS_Read.Variable.DistanceCalculation )
      wire#w1
      Contact( "DB7259_UNIT_03_STA_MEAS_B_ENABLE_DISABLE".ENABLED )
      wire#w2
      Coil( "DB16000_OPC_UA_TRIGGER_ALARM".CLIENT.U03_MEAS_STA_MEAS_B.ALARMS.DISTANCE_CALCULATION_A )
   END_RUNG
   RUNG wire#powerrail
      Contact( "DB16000_OPC_UA_TRIGGER_ALARM".CLIENT.U03_MEAS_STA_MEAS_B.ALARMS.DISTANCE_CALCULATION_A )
      I_Contact( "DB2120_MPP_ITC_IPC".RESET_FAULTS )
      I_Contact( "DB7300_INTERLOCK_GENERAL".GENERAL_MACHINE.FROM_CELL_TO_MACHINE_GENERAL.CELL_MEAS_STA_RESET )
   END_RUNG wire#w1
   RUNG wire#w2
      Coil( "DB426_ALARMS_WARNINGS".UNIT_03."724532" )
   END_RUNG
   // the same network as SCL:
   "DB16000_OPC_UA_TRIGGER_ALARM".CLIENT.U03_MEAS_STA_MEAS_B.ALARMS.DISTANCE_CALCULATION_A := ((("DB16007_U03_MEAS_STA_MEAS_B_CLIENT_INTERFACE".U03_FACE_B_MEAS_Read.Variable.Status = (-1)) AND "DB16007_U03_MEAS_STA_MEAS_B_CLIENT_INTERFACE".U03_FACE_B_MEAS_Read.Variable.DistanceCalculation) OR ("DB16000_OPC_UA_TRIGGER_ALARM".CLIENT.U03_MEAS_STA_MEAS_B.ALARMS.DISTANCE_CALCULATION_A AND NOT "DB2120_MPP_ITC_IPC".RESET_FAULTS AND NOT "DB7300_INTERLOCK_GENERAL".GENERAL_MACHINE.FROM_CELL_TO_MACHINE_GENERAL.CELL_MEAS_STA_RESET)) AND "DB7259_UNIT_03_STA_MEAS_B_ENABLE_DISABLE".ENABLED;
   "DB426_ALARMS_WARNINGS".UNIT_03."724532" := "DB16000_OPC_UA_TRIGGER_ALARM".CLIENT.U03_MEAS_STA_MEAS_B.ALARMS.DISTANCE_CALCULATION_A;
END_REGION

REGION Network 30: UNIT 03 MEASURING STATION FACE B LAYER GROWTH ANALYSIS ALARM
   RUNG wire#powerrail
      { S7_Templates := "SrcType := Int" } EQ_Contact(in1 := "DB16007_U03_MEAS_STA_MEAS_B_CLIENT_INTERFACE".U03_FACE_B_MEAS_Read.Variable.Status, in2 := -1)
      Contact( "M_ZERO" )
      wire#w1
      Contact( "DB7259_UNIT_03_STA_MEAS_B_ENABLE_DISABLE".ENABLED )
      wire#w2
      Coil( "DB16000_OPC_UA_TRIGGER_ALARM".CLIENT.U03_MEAS_STA_MEAS_B.ALARMS.LAYER_GROWTH_A )
   END_RUNG
   RUNG wire#powerrail
      Contact( "DB16000_OPC_UA_TRIGGER_ALARM".CLIENT.U03_MEAS_STA_MEAS_B.ALARMS.LAYER_GROWTH_A )
      I_Contact( "DB2120_MPP_ITC_IPC".RESET_FAULTS )
      I_Contact( "DB7300_INTERLOCK_GENERAL".GENERAL_MACHINE.FROM_CELL_TO_MACHINE_GENERAL.CELL_MEAS_STA_RESET )
   END_RUNG wire#w1
   RUNG wire#w2
      Coil( "DB426_ALARMS_WARNINGS".UNIT_03."724527" )
   END_RUNG
   // the same network as SCL:
   "DB16000_OPC_UA_TRIGGER_ALARM".CLIENT.U03_MEAS_STA_MEAS_B.ALARMS.LAYER_GROWTH_A := ((("DB16007_U03_MEAS_STA_MEAS_B_CLIENT_INTERFACE".U03_FACE_B_MEAS_Read.Variable.Status = (-1)) AND "M_ZERO") OR ("DB16000_OPC_UA_TRIGGER_ALARM".CLIENT.U03_MEAS_STA_MEAS_B.ALARMS.LAYER_GROWTH_A AND NOT "DB2120_MPP_ITC_IPC".RESET_FAULTS AND NOT "DB7300_INTERLOCK_GENERAL".GENERAL_MACHINE.FROM_CELL_TO_MACHINE_GENERAL.CELL_MEAS_STA_RESET)) AND "DB7259_UNIT_03_STA_MEAS_B_ENABLE_DISABLE".ENABLED;
   "DB426_ALARMS_WARNINGS".UNIT_03."724527" := "DB16000_OPC_UA_TRIGGER_ALARM".CLIENT.U03_MEAS_STA_MEAS_B.ALARMS.LAYER_GROWTH_A;
END_REGION

REGION Network 31: UNIT 03 MEASURING STATION FACE B SURFACE DEFECTS ANALYSIS ALARM
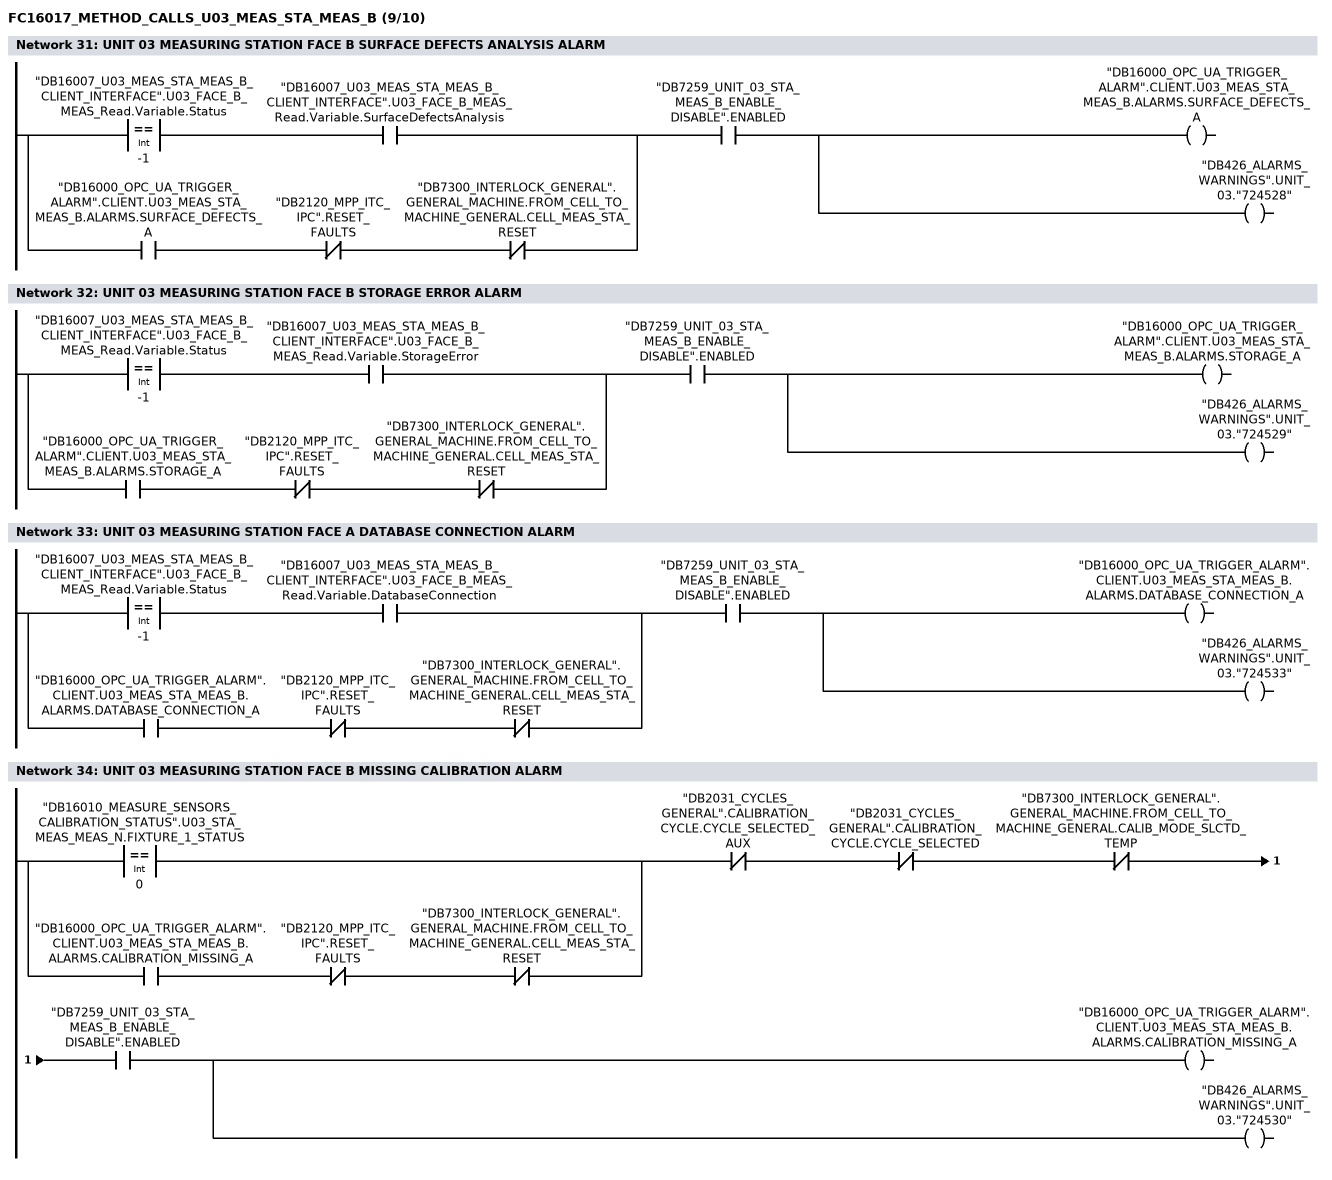
   RUNG wire#powerrail
      { S7_Templates := "SrcType := Int" } EQ_Contact(in1 := "DB16007_U03_MEAS_STA_MEAS_B_CLIENT_INTERFACE".U03_FACE_B_MEAS_Read.Variable.Status, in2 := -1)
      Contact( "DB16007_U03_MEAS_STA_MEAS_B_CLIENT_INTERFACE".U03_FACE_B_MEAS_Read.Variable.SurfaceDefectsAnalysis )
      wire#w1
      Contact( "DB7259_UNIT_03_STA_MEAS_B_ENABLE_DISABLE".ENABLED )
      wire#w2
      Coil( "DB16000_OPC_UA_TRIGGER_ALARM".CLIENT.U03_MEAS_STA_MEAS_B.ALARMS.SURFACE_DEFECTS_A )
   END_RUNG
   RUNG wire#powerrail
      Contact( "DB16000_OPC_UA_TRIGGER_ALARM".CLIENT.U03_MEAS_STA_MEAS_B.ALARMS.SURFACE_DEFECTS_A )
      I_Contact( "DB2120_MPP_ITC_IPC".RESET_FAULTS )
      I_Contact( "DB7300_INTERLOCK_GENERAL".GENERAL_MACHINE.FROM_CELL_TO_MACHINE_GENERAL.CELL_MEAS_STA_RESET )
   END_RUNG wire#w1
   RUNG wire#w2
      Coil( "DB426_ALARMS_WARNINGS".UNIT_03."724528" )
   END_RUNG
   // the same network as SCL:
   "DB16000_OPC_UA_TRIGGER_ALARM".CLIENT.U03_MEAS_STA_MEAS_B.ALARMS.SURFACE_DEFECTS_A := ((("DB16007_U03_MEAS_STA_MEAS_B_CLIENT_INTERFACE".U03_FACE_B_MEAS_Read.Variable.Status = (-1)) AND "DB16007_U03_MEAS_STA_MEAS_B_CLIENT_INTERFACE".U03_FACE_B_MEAS_Read.Variable.SurfaceDefectsAnalysis) OR ("DB16000_OPC_UA_TRIGGER_ALARM".CLIENT.U03_MEAS_STA_MEAS_B.ALARMS.SURFACE_DEFECTS_A AND NOT "DB2120_MPP_ITC_IPC".RESET_FAULTS AND NOT "DB7300_INTERLOCK_GENERAL".GENERAL_MACHINE.FROM_CELL_TO_MACHINE_GENERAL.CELL_MEAS_STA_RESET)) AND "DB7259_UNIT_03_STA_MEAS_B_ENABLE_DISABLE".ENABLED;
   "DB426_ALARMS_WARNINGS".UNIT_03."724528" := "DB16000_OPC_UA_TRIGGER_ALARM".CLIENT.U03_MEAS_STA_MEAS_B.ALARMS.SURFACE_DEFECTS_A;
END_REGION

REGION Network 32: UNIT 03 MEASURING STATION FACE B STORAGE ERROR ALARM
   RUNG wire#powerrail
      { S7_Templates := "SrcType := Int" } EQ_Contact(in1 := "DB16007_U03_MEAS_STA_MEAS_B_CLIENT_INTERFACE".U03_FACE_B_MEAS_Read.Variable.Status, in2 := -1)
      Contact( "DB16007_U03_MEAS_STA_MEAS_B_CLIENT_INTERFACE".U03_FACE_B_MEAS_Read.Variable.StorageError )
      wire#w1
      Contact( "DB7259_UNIT_03_STA_MEAS_B_ENABLE_DISABLE".ENABLED )
      wire#w2
      Coil( "DB16000_OPC_UA_TRIGGER_ALARM".CLIENT.U03_MEAS_STA_MEAS_B.ALARMS.STORAGE_A )
   END_RUNG
   RUNG wire#powerrail
      Contact( "DB16000_OPC_UA_TRIGGER_ALARM".CLIENT.U03_MEAS_STA_MEAS_B.ALARMS.STORAGE_A )
      I_Contact( "DB2120_MPP_ITC_IPC".RESET_FAULTS )
      I_Contact( "DB7300_INTERLOCK_GENERAL".GENERAL_MACHINE.FROM_CELL_TO_MACHINE_GENERAL.CELL_MEAS_STA_RESET )
   END_RUNG wire#w1
   RUNG wire#w2
      Coil( "DB426_ALARMS_WARNINGS".UNIT_03."724529" )
   END_RUNG
   // the same network as SCL:
   "DB16000_OPC_UA_TRIGGER_ALARM".CLIENT.U03_MEAS_STA_MEAS_B.ALARMS.STORAGE_A := ((("DB16007_U03_MEAS_STA_MEAS_B_CLIENT_INTERFACE".U03_FACE_B_MEAS_Read.Variable.Status = (-1)) AND "DB16007_U03_MEAS_STA_MEAS_B_CLIENT_INTERFACE".U03_FACE_B_MEAS_Read.Variable.StorageError) OR ("DB16000_OPC_UA_TRIGGER_ALARM".CLIENT.U03_MEAS_STA_MEAS_B.ALARMS.STORAGE_A AND NOT "DB2120_MPP_ITC_IPC".RESET_FAULTS AND NOT "DB7300_INTERLOCK_GENERAL".GENERAL_MACHINE.FROM_CELL_TO_MACHINE_GENERAL.CELL_MEAS_STA_RESET)) AND "DB7259_UNIT_03_STA_MEAS_B_ENABLE_DISABLE".ENABLED;
   "DB426_ALARMS_WARNINGS".UNIT_03."724529" := "DB16000_OPC_UA_TRIGGER_ALARM".CLIENT.U03_MEAS_STA_MEAS_B.ALARMS.STORAGE_A;
END_REGION

REGION Network 33: UNIT 03 MEASURING STATION FACE A DATABASE CONNECTION ALARM
   RUNG wire#powerrail
      { S7_Templates := "SrcType := Int" } EQ_Contact(in1 := "DB16007_U03_MEAS_STA_MEAS_B_CLIENT_INTERFACE".U03_FACE_B_MEAS_Read.Variable.Status, in2 := -1)
      Contact( "DB16007_U03_MEAS_STA_MEAS_B_CLIENT_INTERFACE".U03_FACE_B_MEAS_Read.Variable.DatabaseConnection )
      wire#w1
      Contact( "DB7259_UNIT_03_STA_MEAS_B_ENABLE_DISABLE".ENABLED )
      wire#w2
      Coil( "DB16000_OPC_UA_TRIGGER_ALARM".CLIENT.U03_MEAS_STA_MEAS_B.ALARMS.DATABASE_CONNECTION_A )
   END_RUNG
   RUNG wire#powerrail
      Contact( "DB16000_OPC_UA_TRIGGER_ALARM".CLIENT.U03_MEAS_STA_MEAS_B.ALARMS.DATABASE_CONNECTION_A )
      I_Contact( "DB2120_MPP_ITC_IPC".RESET_FAULTS )
      I_Contact( "DB7300_INTERLOCK_GENERAL".GENERAL_MACHINE.FROM_CELL_TO_MACHINE_GENERAL.CELL_MEAS_STA_RESET )
   END_RUNG wire#w1
   RUNG wire#w2
      Coil( "DB426_ALARMS_WARNINGS".UNIT_03."724533" )
   END_RUNG
   // the same network as SCL:
   "DB16000_OPC_UA_TRIGGER_ALARM".CLIENT.U03_MEAS_STA_MEAS_B.ALARMS.DATABASE_CONNECTION_A := ((("DB16007_U03_MEAS_STA_MEAS_B_CLIENT_INTERFACE".U03_FACE_B_MEAS_Read.Variable.Status = (-1)) AND "DB16007_U03_MEAS_STA_MEAS_B_CLIENT_INTERFACE".U03_FACE_B_MEAS_Read.Variable.DatabaseConnection) OR ("DB16000_OPC_UA_TRIGGER_ALARM".CLIENT.U03_MEAS_STA_MEAS_B.ALARMS.DATABASE_CONNECTION_A AND NOT "DB2120_MPP_ITC_IPC".RESET_FAULTS AND NOT "DB7300_INTERLOCK_GENERAL".GENERAL_MACHINE.FROM_CELL_TO_MACHINE_GENERAL.CELL_MEAS_STA_RESET)) AND "DB7259_UNIT_03_STA_MEAS_B_ENABLE_DISABLE".ENABLED;
   "DB426_ALARMS_WARNINGS".UNIT_03."724533" := "DB16000_OPC_UA_TRIGGER_ALARM".CLIENT.U03_MEAS_STA_MEAS_B.ALARMS.DATABASE_CONNECTION_A;
END_REGION

REGION Network 34: UNIT 03 MEASURING STATION FACE B MISSING CALIBRATION ALARM
   RUNG wire#powerrail
      { S7_Templates := "SrcType := Int" } EQ_Contact(in1 := "DB16010_MEASURE_SENSORS_CALIBRATION_STATUS".U03_STA_MEAS_MEAS_N.FIXTURE_1_STATUS, in2 := 0)
      wire#w1
      I_Contact( "DB2031_CYCLES_GENERAL".CALIBRATION_CYCLE.CYCLE_SELECTED_AUX )
      I_Contact( "DB2031_CYCLES_GENERAL".CALIBRATION_CYCLE.CYCLE_SELECTED )
      I_Contact( "DB7300_INTERLOCK_GENERAL".GENERAL_MACHINE.FROM_CELL_TO_MACHINE_GENERAL.CALIB_MODE_SLCTD_TEMP )
      Contact( "DB7259_UNIT_03_STA_MEAS_B_ENABLE_DISABLE".ENABLED )
      wire#w2
      Coil( "DB16000_OPC_UA_TRIGGER_ALARM".CLIENT.U03_MEAS_STA_MEAS_B.ALARMS.CALIBRATION_MISSING_A )
   END_RUNG
   RUNG wire#powerrail
      Contact( "DB16000_OPC_UA_TRIGGER_ALARM".CLIENT.U03_MEAS_STA_MEAS_B.ALARMS.CALIBRATION_MISSING_A )
      I_Contact( "DB2120_MPP_ITC_IPC".RESET_FAULTS )
      I_Contact( "DB7300_INTERLOCK_GENERAL".GENERAL_MACHINE.FROM_CELL_TO_MACHINE_GENERAL.CELL_MEAS_STA_RESET )
   END_RUNG wire#w1
   RUNG wire#w2
      Coil( "DB426_ALARMS_WARNINGS".UNIT_03."724530" )
   END_RUNG
   // the same network as SCL:
   "DB16000_OPC_UA_TRIGGER_ALARM".CLIENT.U03_MEAS_STA_MEAS_B.ALARMS.CALIBRATION_MISSING_A := (("DB16010_MEASURE_SENSORS_CALIBRATION_STATUS".U03_STA_MEAS_MEAS_N.FIXTURE_1_STATUS = 0) OR ("DB16000_OPC_UA_TRIGGER_ALARM".CLIENT.U03_MEAS_STA_MEAS_B.ALARMS.CALIBRATION_MISSING_A AND NOT "DB2120_MPP_ITC_IPC".RESET_FAULTS AND NOT "DB7300_INTERLOCK_GENERAL".GENERAL_MACHINE.FROM_CELL_TO_MACHINE_GENERAL.CELL_MEAS_STA_RESET)) AND NOT "DB2031_CYCLES_GENERAL".CALIBRATION_CYCLE.CYCLE_SELECTED_AUX AND NOT "DB2031_CYCLES_GENERAL".CALIBRATION_CYCLE.CYCLE_SELECTED AND NOT "DB7300_INTERLOCK_GENERAL".GENERAL_MACHINE.FROM_CELL_TO_MACHINE_GENERAL.CALIB_MODE_SLCTD_TEMP AND "DB7259_UNIT_03_STA_MEAS_B_ENABLE_DISABLE".ENABLED;
   "DB426_ALARMS_WARNINGS".UNIT_03."724530" := "DB16000_OPC_UA_TRIGGER_ALARM".CLIENT.U03_MEAS_STA_MEAS_B.ALARMS.CALIBRATION_MISSING_A;
END_REGION

REGION Network 35: UNIT 03 MEASURING STATION FACE B CALIBRATION PROCEDURE ALARM
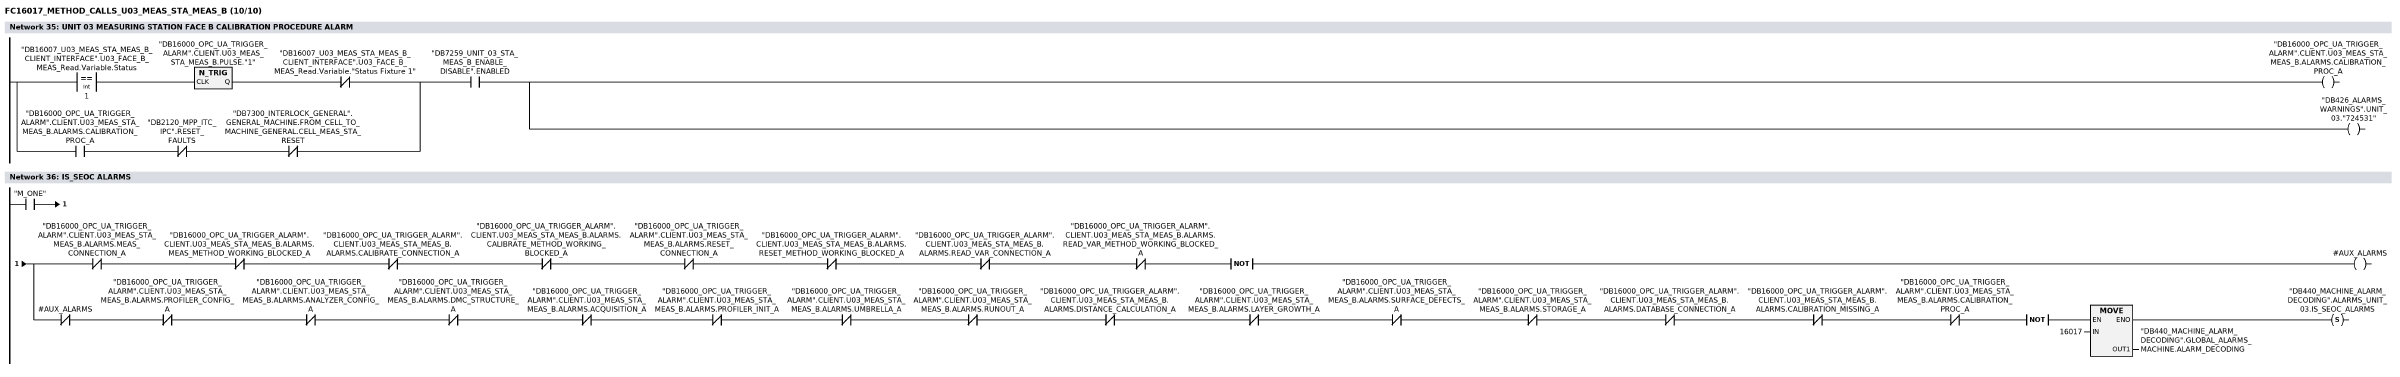
   RUNG wire#powerrail
      { S7_Templates := "SrcType := Int" } EQ_Contact(in1 := "DB16007_U03_MEAS_STA_MEAS_B_CLIENT_INTERFACE".U03_FACE_B_MEAS_Read.Variable.Status, in2 := 1)
      N_Trig( "DB16000_OPC_UA_TRIGGER_ALARM".CLIENT.U03_MEAS_STA_MEAS_B.PULSE."1" )
      I_Contact( "DB16007_U03_MEAS_STA_MEAS_B_CLIENT_INTERFACE".U03_FACE_B_MEAS_Read.Variable."Status Fixture 1" )
      wire#w1
      Contact( "DB7259_UNIT_03_STA_MEAS_B_ENABLE_DISABLE".ENABLED )
      wire#w2
      Coil( "DB16000_OPC_UA_TRIGGER_ALARM".CLIENT.U03_MEAS_STA_MEAS_B.ALARMS.CALIBRATION_PROC_A )
   END_RUNG
   RUNG wire#powerrail
      Contact( "DB16000_OPC_UA_TRIGGER_ALARM".CLIENT.U03_MEAS_STA_MEAS_B.ALARMS.CALIBRATION_PROC_A )
      I_Contact( "DB2120_MPP_ITC_IPC".RESET_FAULTS )
      I_Contact( "DB7300_INTERLOCK_GENERAL".GENERAL_MACHINE.FROM_CELL_TO_MACHINE_GENERAL.CELL_MEAS_STA_RESET )
   END_RUNG wire#w1
   RUNG wire#w2
      Coil( "DB426_ALARMS_WARNINGS".UNIT_03."724531" )
   END_RUNG
   // the same network as SCL:
   #_w1 := "DB16007_U03_MEAS_STA_MEAS_B_CLIENT_INTERFACE".U03_FACE_B_MEAS_Read.Variable.Status = 1;
   #_w2 := NOT #_w1 AND "DB16000_OPC_UA_TRIGGER_ALARM".CLIENT.U03_MEAS_STA_MEAS_B.PULSE."1";   // falling edge
   "DB16000_OPC_UA_TRIGGER_ALARM".CLIENT.U03_MEAS_STA_MEAS_B.PULSE."1" := #_w1;
   "DB16000_OPC_UA_TRIGGER_ALARM".CLIENT.U03_MEAS_STA_MEAS_B.ALARMS.CALIBRATION_PROC_A := ((#_w2 AND NOT "DB16007_U03_MEAS_STA_MEAS_B_CLIENT_INTERFACE".U03_FACE_B_MEAS_Read.Variable."Status Fixture 1") OR ("DB16000_OPC_UA_TRIGGER_ALARM".CLIENT.U03_MEAS_STA_MEAS_B.ALARMS.CALIBRATION_PROC_A AND NOT "DB2120_MPP_ITC_IPC".RESET_FAULTS AND NOT "DB7300_INTERLOCK_GENERAL".GENERAL_MACHINE.FROM_CELL_TO_MACHINE_GENERAL.CELL_MEAS_STA_RESET)) AND "DB7259_UNIT_03_STA_MEAS_B_ENABLE_DISABLE".ENABLED;
   "DB426_ALARMS_WARNINGS".UNIT_03."724531" := "DB16000_OPC_UA_TRIGGER_ALARM".CLIENT.U03_MEAS_STA_MEAS_B.ALARMS.CALIBRATION_PROC_A;
END_REGION

REGION Network 36: IS_SEOC ALARMS
   RUNG wire#powerrail
      Contact( "M_ONE" )
      wire#w1
      I_Contact( "DB16000_OPC_UA_TRIGGER_ALARM".CLIENT.U03_MEAS_STA_MEAS_B.ALARMS.MEAS_CONNECTION_A )
      I_Contact( "DB16000_OPC_UA_TRIGGER_ALARM".CLIENT.U03_MEAS_STA_MEAS_B.ALARMS.MEAS_METHOD_WORKING_BLOCKED_A )
      I_Contact( "DB16000_OPC_UA_TRIGGER_ALARM".CLIENT.U03_MEAS_STA_MEAS_B.ALARMS.CALIBRATE_CONNECTION_A )
      I_Contact( "DB16000_OPC_UA_TRIGGER_ALARM".CLIENT.U03_MEAS_STA_MEAS_B.ALARMS.CALIBRATE_METHOD_WORKING_BLOCKED_A )
      I_Contact( "DB16000_OPC_UA_TRIGGER_ALARM".CLIENT.U03_MEAS_STA_MEAS_B.ALARMS.RESET_CONNECTION_A )
      I_Contact( "DB16000_OPC_UA_TRIGGER_ALARM".CLIENT.U03_MEAS_STA_MEAS_B.ALARMS.RESET_METHOD_WORKING_BLOCKED_A )
      I_Contact( "DB16000_OPC_UA_TRIGGER_ALARM".CLIENT.U03_MEAS_STA_MEAS_B.ALARMS.READ_VAR_CONNECTION_A )
      I_Contact( "DB16000_OPC_UA_TRIGGER_ALARM".CLIENT.U03_MEAS_STA_MEAS_B.ALARMS.READ_VAR_METHOD_WORKING_BLOCKED_A )
      Not()
      Coil( #AUX_ALARMS )
   END_RUNG
   RUNG wire#w1
      I_Contact( #AUX_ALARMS )
      I_Contact( "DB16000_OPC_UA_TRIGGER_ALARM".CLIENT.U03_MEAS_STA_MEAS_B.ALARMS.PROFILER_CONFIG_A )
      I_Contact( "DB16000_OPC_UA_TRIGGER_ALARM".CLIENT.U03_MEAS_STA_MEAS_B.ALARMS.ANALYZER_CONFIG_A )
      I_Contact( "DB16000_OPC_UA_TRIGGER_ALARM".CLIENT.U03_MEAS_STA_MEAS_B.ALARMS.DMC_STRUCTURE_A )
      I_Contact( "DB16000_OPC_UA_TRIGGER_ALARM".CLIENT.U03_MEAS_STA_MEAS_B.ALARMS.ACQUISITION_A )
      I_Contact( "DB16000_OPC_UA_TRIGGER_ALARM".CLIENT.U03_MEAS_STA_MEAS_B.ALARMS.PROFILER_INIT_A )
      I_Contact( "DB16000_OPC_UA_TRIGGER_ALARM".CLIENT.U03_MEAS_STA_MEAS_B.ALARMS.UMBRELLA_A )
      I_Contact( "DB16000_OPC_UA_TRIGGER_ALARM".CLIENT.U03_MEAS_STA_MEAS_B.ALARMS.RUNOUT_A )
      I_Contact( "DB16000_OPC_UA_TRIGGER_ALARM".CLIENT.U03_MEAS_STA_MEAS_B.ALARMS.DISTANCE_CALCULATION_A )
      I_Contact( "DB16000_OPC_UA_TRIGGER_ALARM".CLIENT.U03_MEAS_STA_MEAS_B.ALARMS.LAYER_GROWTH_A )
      I_Contact( "DB16000_OPC_UA_TRIGGER_ALARM".CLIENT.U03_MEAS_STA_MEAS_B.ALARMS.SURFACE_DEFECTS_A )
      I_Contact( "DB16000_OPC_UA_TRIGGER_ALARM".CLIENT.U03_MEAS_STA_MEAS_B.ALARMS.STORAGE_A )
      I_Contact( "DB16000_OPC_UA_TRIGGER_ALARM".CLIENT.U03_MEAS_STA_MEAS_B.ALARMS.DATABASE_CONNECTION_A )
      I_Contact( "DB16000_OPC_UA_TRIGGER_ALARM".CLIENT.U03_MEAS_STA_MEAS_B.ALARMS.CALIBRATION_MISSING_A )
      I_Contact( "DB16000_OPC_UA_TRIGGER_ALARM".CLIENT.U03_MEAS_STA_MEAS_B.ALARMS.CALIBRATION_PROC_A )
      Not()
      Move(in := 16017, out1 => "DB440_MACHINE_ALARM_DECODING".GLOBAL_ALARMS_MACHINE.ALARM_DECODING)
      S_Coil( "DB440_MACHINE_ALARM_DECODING".ALARMS_UNIT_03.IS_SEOC_ALARMS )
   END_RUNG
   // the same network as SCL:
   #AUX_ALARMS := NOT ("M_ONE" AND NOT "DB16000_OPC_UA_TRIGGER_ALARM".CLIENT.U03_MEAS_STA_MEAS_B.ALARMS.MEAS_CONNECTION_A AND NOT "DB16000_OPC_UA_TRIGGER_ALARM".CLIENT.U03_MEAS_STA_MEAS_B.ALARMS.MEAS_METHOD_WORKING_BLOCKED_A AND NOT "DB16000_OPC_UA_TRIGGER_ALARM".CLIENT.U03_MEAS_STA_MEAS_B.ALARMS.CALIBRATE_CONNECTION_A AND NOT "DB16000_OPC_UA_TRIGGER_ALARM".CLIENT.U03_MEAS_STA_MEAS_B.ALARMS.CALIBRATE_METHOD_WORKING_BLOCKED_A AND NOT "DB16000_OPC_UA_TRIGGER_ALARM".CLIENT.U03_MEAS_STA_MEAS_B.ALARMS.RESET_CONNECTION_A AND NOT "DB16000_OPC_UA_TRIGGER_ALARM".CLIENT.U03_MEAS_STA_MEAS_B.ALARMS.RESET_METHOD_WORKING_BLOCKED_A AND NOT "DB16000_OPC_UA_TRIGGER_ALARM".CLIENT.U03_MEAS_STA_MEAS_B.ALARMS.READ_VAR_CONNECTION_A AND NOT "DB16000_OPC_UA_TRIGGER_ALARM".CLIENT.U03_MEAS_STA_MEAS_B.ALARMS.READ_VAR_METHOD_WORKING_BLOCKED_A);
   IF NOT ("M_ONE" AND NOT #AUX_ALARMS AND NOT "DB16000_OPC_UA_TRIGGER_ALARM".CLIENT.U03_MEAS_STA_MEAS_B.ALARMS.PROFILER_CONFIG_A AND NOT "DB16000_OPC_UA_TRIGGER_ALARM".CLIENT.U03_MEAS_STA_MEAS_B.ALARMS.ANALYZER_CONFIG_A AND NOT "DB16000_OPC_UA_TRIGGER_ALARM".CLIENT.U03_MEAS_STA_MEAS_B.ALARMS.DMC_STRUCTURE_A AND NOT "DB16000_OPC_UA_TRIGGER_ALARM".CLIENT.U03_MEAS_STA_MEAS_B.ALARMS.ACQUISITION_A AND NOT "DB16000_OPC_UA_TRIGGER_ALARM".CLIENT.U03_MEAS_STA_MEAS_B.ALARMS.PROFILER_INIT_A AND NOT "DB16000_OPC_UA_TRIGGER_ALARM".CLIENT.U03_MEAS_STA_MEAS_B.ALARMS.UMBRELLA_A AND NOT "DB16000_OPC_UA_TRIGGER_ALARM".CLIENT.U03_MEAS_STA_MEAS_B.ALARMS.RUNOUT_A AND NOT "DB16000_OPC_UA_TRIGGER_ALARM".CLIENT.U03_MEAS_STA_MEAS_B.ALARMS.DISTANCE_CALCULATION_A AND NOT "DB16000_OPC_UA_TRIGGER_ALARM".CLIENT.U03_MEAS_STA_MEAS_B.ALARMS.LAYER_GROWTH_A AND NOT "DB16000_OPC_UA_TRIGGER_ALARM".CLIENT.U03_MEAS_STA_MEAS_B.ALARMS.SURFACE_DEFECTS_A AND NOT "DB16000_OPC_UA_TRIGGER_ALARM".CLIENT.U03_MEAS_STA_MEAS_B.ALARMS.STORAGE_A AND NOT "DB16000_OPC_UA_TRIGGER_ALARM".CLIENT.U03_MEAS_STA_MEAS_B.ALARMS.DATABASE_CONNECTION_A AND NOT "DB16000_OPC_UA_TRIGGER_ALARM".CLIENT.U03_MEAS_STA_MEAS_B.ALARMS.CALIBRATION_MISSING_A AND NOT "DB16000_OPC_UA_TRIGGER_ALARM".CLIENT.U03_MEAS_STA_MEAS_B.ALARMS.CALIBRATION_PROC_A) THEN
       "DB440_MACHINE_ALARM_DECODING".GLOBAL_ALARMS_MACHINE.ALARM_DECODING := 16017;
       "DB440_MACHINE_ALARM_DECODING".ALARMS_UNIT_03.IS_SEOC_ALARMS := TRUE;
   END_IF;
END_REGION
END_FUNCTION
